	{region "============= 進到設定位置  ============="}
	40: // 判斷前進後退
		IF BD_moveDis - FxB_Clamp_Pos > 0 THEN
			// 目標大於現在位置
			o_BD_Clamp_Close	:= FALSE;
			o_BD_Clamp_Open		:= TRUE;
			step_BD_C.Step  := step_BD_C.Step  + 1;
		ELSIF BD_moveDis - FxB_Clamp_Pos < 0 THEN
			// 目標小於現在位置
			o_BD_Clamp_Close	:= TRUE;
			o_BD_Clamp_Open		:= FALSE;
			step_BD_C.Step  := step_BD_C.Step  + 1;
		ELSE
			step_BD_C.Step  := 90;
		END_IF
		
	41: // 設定位置 - 目前位置 (接近0表示位置到達) <= 停止位移補償(移動速度 * 停止時間) 
		IF ABS(BD_moveDis - FxB_Clamp_Pos) <= (ABS(FxB_Clamp_Spd) * 0.1) THEN
			o_BD_Clamp_Close		:= FALSE;
			o_BD_Clamp_Open		:= FALSE;
			step_BD_C.Step  := step_BD_C.Step  + 1;
		END_IF
		
		// 靜止1秒後，標示為功能完成
		tmr106.IN := ABS(FxB_Clamp_Spd) <= 1;
		tmr106.PT := T#1S;
		IF tmr106.Q THEN
			tmr106.IN := FALSE;
			step_BD_C.Step  := step_BD_C.Step  + 1;
		END_IF
			 
	42:
		o_BD_Clamp_Open		:= FALSE;
		o_BD_Clamp_Close	:= FALSE;
		step_BD_C.Step  := step_BD_C.Step  + 1;
			 
	43:
		 step_BD_C.Step  := 90;
	
{endregion}
		
	90:
		BD_moveDis := 0;
		step_BD_C.bDone := TRUE;
		step_BD_C.Step  := 0;
END_CASE

IF o_BD_Clamp_Open THEN
	b_BD_Clamp := FALSE;
END_IF

step_BD_C.bBuzy := step_BD_C.Step > 0 AND step_BD_C.Step < 10000;
step_BD_C.bError := step_BD_C.Step >= 10000;

IF step_BD_C.bError OR step_BD_C.bBuzy THEN
	step_BD_C.bDone := FALSE;
END_IF
END_ACTION

ACTION Step_BD_01_UnClamp:
CASE step_BD_C.Step  OF
	// FxA動作前檢查檢查
	100: // 檢查Group B Z軸位置，需在桁架中間 (Z pos > 500 )
		tmr01.IN := FALSE;
		IF GbZ.pos > 500 OR GbX.fPos < 50 OR NOT Hmi.Jog_UnLimite THEN
			step_BD_C.Step  := step_BD_C.Step  + 1;
		ELSE
			step_BD_C.Step  := step_BD_C.Step  + 10000;
			strmem1.WRITE(name);
			strmem1.APPEND(":Group B 位置錯誤,再非安全位置:");
			strmem1.APPEND(STR := WCONCAT("(X:", TO_WSTRING(GbX.pos)));
			strmem1.APPEND(STR := WCONCAT(",Y:", TO_WSTRING(GbY.pos)));
			strmem1.APPEND(STR := WCONCAT(",Z:", TO_WSTRING(GbZ.pos)));
			strmem1.APPEND(")");
			pMsg.Push_Error(strmem1.READ);
		END_IF
		
	101: 
		IF o_Oil_Pressure_Pump THEN
			step_BD_C.Step  := step_BD_C.Step  + 1;
		END_IF
		
	102:
		step_BD_C.Step  := 110;
	
		// 確認BD下壓位置
//		IF pressureB_home_sensor AND pressureD_home_sensor THEN
//			step_BD_C.Step  := step_BD_C.Step  + 1;
//		ELSE
//			step_BD_C.Step  := step_BD_C.Step  + 10000;
//			pMsg.Push_Error(StrConcat_2(name, ":下壓B or 下壓D 未停在原點，動作取消 "));
//		END_IF
		
		
		
	110: // 放開選擇
		o_BD_Encoder_enable		:= FALSE;
		o_BD_Encoder_disable	:= TRUE;
		IF BD_moveDis = 0 THEN
			// 退到原點
			step_BD_C.Step  := 120; 
		ELSE
			// 退到設定距離
			step_BD_C.Step  := 140;
		END_IF

	{region "============= 退到原點  ============="}
	120: // 放開BD夾輪夾
		o_BD_Clamp_Close	:= FALSE;
		o_BD_Clamp_Open		:= TRUE;
		step_BD_C.Step  := step_BD_C.Step  + 1;
		
	121: // 確定BD夾輪停止移動
		tmr106.IN := ABS(FxB_Clamp_Spd) <= 1 ;
		tmr106.PT := T#1S;
		IF tmr106.Q THEN
			tmr106.IN := FALSE;
			step_BD_C.Step  := step_BD_C.Step  + 1;
		END_IF
		
	122:
		o_BD_Clamp_Open		:= FALSE;
		step_BD_C.Step  := step_BD_C.Step  + 1;
		
	123: 
		step_BD_C.Step  := 130;
		
	130:
		step_BD_C.Step  := 190;
	{endregion}		
		
		
		
	{region "============= 退到設定距離  ============="}
	140: // 紀錄開始位置
		BD_StartPos := FxB_Clamp_Pos;
		step_BD_C.Step  := step_BD_C.Step  + 1;
		
	141: // 開始後退
		o_BD_Clamp_Close	:= FALSE;
		o_BD_Clamp_Open		:= TRUE;
		step_BD_C.Step := step_BD_C.step + 1;
		
	142: // 大於設定距離
		IF ABS(BD_StartPos - FxB_Clamp_Pos)  >= ABS(BD_moveDis) - ( ABS(FxB_Clamp_Spd) * 0.1) THEN
			o_BD_Clamp_Open		:= FALSE;
			step_BD_C.step := step_BD_C.step + 1;
		END_IF
		
		tmr106.IN := ABS(FxB_Clamp_Spd) <= 1 ;
		tmr106.PT := T#1S;
		IF tmr01.Q THEN
			tmr106.IN := FALSE;
			step_BD_C.Step  := step_BD_C.Step  + 1;
		END_IF
			 
	143:
		o_BD_Clamp_Open		:= FALSE;
		o_BD_Clamp_Close	:= FALSE;
		step_BD_C.step := step_BD_C.step + 1;
			 
	144:
		 step_BD_C.step := 190;
	
	{endregion}
	190:
		o_BD_Encoder_enable		:= FALSE;
		o_BD_Encoder_disable	:= FALSE;
		o_BD_Clamp_Open		:= FALSE;
		step_BD_C.bDone := TRUE;
		step_BD_C.step := 0;
END_CASE
END_ACTION

ACTION Step_BD_02_Stop:
CASE step_BD_C.step OF
	// FxA動作前檢查檢查
	200: 
		step_BD_C.step := 210;
		
		
	210: // BD夾輪夾
		o_BD_Clamp_Open		:= FALSE;
		o_BD_Clamp_Close	:= FALSE;
		step_BD_C.step := step_BD_C.step + 1;
		
	211: 
		step_BD_C.step := 0;
END_CASE
END_ACTION

ACTION Step_BD_03_Home:
CASE step_BD_C.Step  OF
	// FxA動作前檢查檢查
	300:  // 檢查Group B Z軸位置，需在桁架中間 (Z pos > 500 )
		tmr01.IN := FALSE;
		Axis.Encoder_FxA_Clamp.MDP5001_511_Output.MDP5001_511_Control.Set_counter_on_latch_C := FALSE;
		Axis.Encoder_FxA_Clamp.MDP5001_511_Output.MDP5001_511_Control.Set_counter := FALSE;
		IF GbZ.fPos >= 490 OR GbX.fPos < 50 OR Hmi.Jog_UnLimite THEN
			step_BD_C.Step  := step_BD_C.Step  + 1;
		ELSE
			step_BD_C.Step  := step_BD_C.Step  + 20000;
			strmem1.WRITE(name);
			strmem1.APPEND(":Group B 位置錯誤,再非安全位置:");
			strmem1.APPEND(STR := WCONCAT("(X:", TO_WSTRING(GbX.pos)));
			strmem1.APPEND(STR := WCONCAT(",Y:", TO_WSTRING(GbY.pos)));
			strmem1.APPEND(STR := WCONCAT(",Z:", TO_WSTRING(GbZ.pos)));
			strmem1.APPEND(")");
			pMsg.Push_Error(strmem1.READ);
		END_IF
		
		// 確認AC下壓位置
//		IF pressureA_home_sensor AND pressureC_home_sensor THEN
//			step_BD_C.Step  := step_BD_C.Step  + 1;
//		ELSE
//			step_BD_C.Step  := step_BD_C.Step  + 10000;
//			pMsg.Push_Error(StrConcat_2(name, ":下壓A or 下壓C 未停在原點，動作取消 "));
//		END_IF
		
	301: 
		IF o_Oil_Pressure_Pump THEN
			step_BD_C.Step  := step_BD_C.Step  + 1;
		END_IF
		
	302:
		IF IO.i510 THEN
			step_BD_C.Step  := 310; 
		ELSE
			step_BD_C.Step  := 320; 
		END_IF
		
		
		
	310: // AC夾輪夾
		o_BD_Clamp_Open		:= TRUE;
		o_BD_Clamp_Close	:= FALSE;
		step_BD_C.Step  := step_BD_C.Step  + 1;
		
	311:
		tmr106.IN := NOT IO.i510;
		tmr106.PT := T#1S;
		IF tmr106.Q THEN
			tmr106.IN := FALSE;
			step_BD_C.Step  := step_BD_C.Step  + 1;
		END_IF
		
	312:
		o_BD_Clamp_Open		:= FALSE;
		o_BD_Clamp_Close	:= FALSE;
		step_BD_C.Step  := step_BD_C.Step  + 1;
		
	313:
		step_BD_C.Step  := 320;
		
		
	320:
		Axis.Encoder_FxB_Clamp.MDP5001_511_Output.MDP5001_511_Control.Set_counter_on_latch_C := TRUE;
		Axis.Encoder_FxB_Clamp.MDP5001_511_Output.MDP5001_511_Set_counter_value := 10000;
		step_BD_C.Step  := step_BD_C.Step  + 1;
		
	321:
		o_BD_Clamp_Open		:= FALSE;
		o_BD_Clamp_Close	:= TRUE;
		step_BD_C.Step  := step_BD_C.Step  + 1;
			
	322:
		// 編碼器歸零完成
		IF Axis.Encoder_FxB_Clamp.MDP5001_511_Input.MDP5001_511_Status.Set_counter_done THEN
			Axis.Encoder_FxB_Clamp.MDP5001_511_Output.MDP5001_511_Control.Set_counter_on_latch_C := FALSE;
			b_BD_HOME := TRUE;
			step_BD_C.Step  := step_BD_C.Step  + 1;
		END_IF

	323:
		o_BD_Clamp_Open		:= FALSE;
		o_BD_Clamp_Close	:= FALSE;
		step_BD_C.Step  := step_BD_C.Step  + 1;
		
		
	324:
		step_BD_C.Step  := 330;
	
	330:
		o_BD_Clamp_Open		:= TRUE;
		o_BD_Clamp_Close	:= FALSE;
		step_BD_C.Step  := step_BD_C.Step  + 1;
		
	331:
		tmr106.IN := NOT IO.i510;
		tmr106.PT := T#1S;
		IF tmr106.Q THEN
			tmr106.IN := FALSE;
			step_BD_C.Step  := step_BD_C.Step  + 1;
		END_IF
		
	332:
		o_BD_Clamp_Open		:= FALSE;
		o_BD_Clamp_Close	:= FALSE;
		step_BD_C.Step  := step_BD_C.Step  + 1;
		
	333:
		step_BD_C.bDone := TRUE;
		step_BD_C.Step  := 0;
		
END_CASE
END_ACTION

ACTION Step_C_Push_UnPush:
CASE step_C_P.Step OF
(*	================================
				C下壓
 	================================*)	

	// FxA動作前檢查檢查
	1: // 檢查Group B Z軸位置，需在桁架中間 (Z pos > 500 )
		step_C_P.Step  := step_C_P.Step  + 1;
// 		IF GbZ.fPos >= 495 OR GbX.fPos > 50 OR Hmi.Jog_UnLimite THEN
// 			step_C_P.Step  := step_C_P.Step  + 1;
// 		ELSE
// 			step_C_P.Step  := step_C_P.Step  + 10000;
// 			strmem1.WRITE(name);
// 			strmem1.APPEND(".C_Push");
// 			strmem1.APPEND(":Group B 位置錯誤,再非安全位置:");
// 			strmem1.APPEND(STR := WCONCAT("(X:", TO_WSTRING(GbX.pos)));
// 			strmem1.APPEND(STR := WCONCAT(",Y:", TO_WSTRING(GbY.pos)));
// 			strmem1.APPEND(STR := WCONCAT(",Z:", TO_WSTRING(GbZ.pos)));
// 			strmem1.APPEND(")");
// 			pMsg.Push_Error(strmem1.READ);
// 		END_IF
		
	2:
		tmr114.IN := TRUE;
		tmr114.PT := T#10S;
		IF o_Oil_Pressure_Pump OR tmr113.Q THEN
			tmr113.IN := FALSE;
			IF o_Oil_Pressure_Pump THEN
				step_C_P.Step  := step_C_P.Step  + 1;
			ELSIF tmr113.Q THEN
				pMsg.Push_Error(WStrConcat(name, ".C_Push:下壓B等待油壓系統啟動逾時"));
				step_C_P.Step  := step_C_P.Step  + 10000;
			END_IF
		END_IF
		
	3:
		tmr103.IN := FALSE;
		tmr113.IN := FALSE;
		step_C_P.Step  := 10;
		
		
	10: // 下壓啟動
		o_PressureC_Up := FALSE;
		o_PressureC_Dn := TRUE;
		step_C_P.Step  := step_C_P.Step  + 1;
		
	11:
		tmr103.IN := TRUE;
		tmr103.PT := T#500MS;
		IF tmr103.q THEN
			tmr103.IN := FALSE;
			step_C_P.Step  := step_C_P.Step  + 1;
		END_IF
		
	12:
// 		o_PressureC_Dn := FALSE;
		step_C_P.Step  := step_C_P.Step  + 1;
		
	13:
		tmr103.IN := pressureC_pressure_sensor;
		tmr103.PT := T#500MS;
		tmr113.IN := TRUE;
		tmr113.PT := T#30S;
		IF tmr103.q OR tmr113.q THEN
			tmr103.IN := FALSE;
			tmr113.IN := FALSE;
			step_C_P.Step  := step_C_P.Step  + 1;
		END_IF
		
	14:
		step_C_P.bDone := TRUE;
		step_C_P.Step  := 0;


(*	================================
				C放開
 	================================*)
	// FxA動作前檢查檢查
	100: // 檢查Group B Z軸位置，需在桁架中間 (Z pos > 500 )
		IF GbZ.pos >= 495 OR GbX.fPos < 50 OR Hmi.Jog_UnLimite OR
			(_C_UnPush_Time > 0 AND _C_UnPush_Time < 10) THEN
			step_C_P.Step  := step_C_P.Step  + 1;
		ELSE
			step_C_P.Step  := step_C_P.Step  + 10000;
			strmem1.WRITE(name);
			strmem1.APPEND(".C_Push");
			strmem1.APPEND(":Group B 位置錯誤,再非安全位置:");
			strmem1.APPEND(STR := WCONCAT("(X:", TO_WSTRING(GbX.pos)));
			strmem1.APPEND(STR := WCONCAT(",Y:", TO_WSTRING(GbY.pos)));
			strmem1.APPEND(STR := WCONCAT(",Z:", TO_WSTRING(GbZ.pos)));
			strmem1.APPEND(")");
			pMsg.Push_Error(strmem1.READ);
		END_IF
		
	101:
		IF o_Oil_Pressure_Pump OR tmr113.Q THEN
			tmr113.IN := FALSE;
			IF o_Oil_Pressure_Pump THEN
				step_C_P.Step  := step_C_P.Step  + 1;
			ELSIF tmr113.Q THEN
				pMsg.Push_Error(WStrConcat(name, ".C_Push:下壓B等待油壓系統啟動逾時"));
				step_C_P.Step  := step_C_P.Step  + 10000;
			END_IF
		END_IF
		
	102:
		tmr103.IN := FALSE;
		tmr113.IN := FALSE;
		step_C_P.Step  := 110;
		
		
	110: // 放開啟動
		o_PressureC_Up := TRUE;
		o_PressureC_Dn := FALSE;
		IF _C_UnPush_Time > 0 THEN
			// 微上升
			step_C_P.Step  := step_C_P.Step  + 20;
		ELSE
			// 升回原點
			step_C_P.Step  := step_C_P.Step  + 10;
		END_IF
		
(*	========================================
					升回原點
	========================================	*)
	120:
		tmr103.IN := TRUE;
		tmr103.PT := T#500MS;
		IF tmr103.q THEN
			tmr103.IN := FALSE;
			step_C_P.Step  := step_C_P.Step  + 1;
		END_IF
		
	121:
// 		o_PressureC_Up := FALSE;
		step_C_P.Step  := step_C_P.Step  + 1;
		
	122:
		tmr103.IN := pressureC_home_sensor;
		tmr103.PT := T#500MS;
		tmr113.IN := TRUE;
		tmr113.PT := T#10S;
		IF tmr103.q OR tmr113.q THEN
			tmr103.IN := FALSE;
			tmr113.IN := FALSE;
			o_PressureC_Up := FALSE;
			step_C_P.Step  := step_C_P.Step  + 1;
		END_IF
		
	123:
		step_C_P.bDone := TRUE;
		step_C_P.Step  := 0;

(*	========================================
					微上升
	========================================	*)
	
	130:
		tmr103.IN := TRUE;
		tmr103.PT := TO_TIME(_C_UnPush_Time * 100);
		IF tmr103.q THEN
			tmr103.IN := FALSE;
			step_C_P.Step  := step_C_P.Step  + 1;
		END_IF
		
	131:
		o_PressureC_Up := FALSE;
		step_C_P.Step  := step_C_P.Step  + 1;
		
	132:
		step_C_P.bDone := TRUE;
		step_C_P.Step  := 0;
	
END_CASE

step_C_P.bBuzy := step_C_P.Step  > 0 AND step_C_P.Step  < 10000;
step_C_P.bError := step_C_P.Step  >= 10000;

IF step_C_P.bBuzy OR step_C_P.bError THEN
	step_C_P.bDone := FALSE;
END_IF
END_ACTION

ACTION Step_D_Push_UnPush:
CASE step_D_P.Step  OF
(*	================================
				D下壓
 	================================*)	

	// FxA動作前檢查檢查
	1: // 檢查Group B Z軸位置，需在桁架中間 (Z pos > 500 )
		IF GbZ.fPos >= 495 OR GbX.fPos < 50 OR Hmi.Jog_UnLimite THEN
			step_D_P.Step  := step_D_P.Step  + 1;
		ELSE
			step_D_P.Step  := step_D_P.Step  + 10000;
			strmem1.WRITE(name);
			strmem1.APPEND(":Group B 位置錯誤,再非安全位置:");
			strmem1.APPEND(STR := WCONCAT("(X:", TO_WSTRING(GbX.pos)));
			strmem1.APPEND(STR := WCONCAT(",Y:", TO_WSTRING(GbY.pos)));
			strmem1.APPEND(STR := WCONCAT(",Z:", TO_WSTRING(GbZ.pos)));
			strmem1.APPEND(")");
			pMsg.Push_Error(strmem1.READ);
		END_IF
		
	2:
		tmr114.IN := TRUE;
		tmr114.PT := T#10S;
		IF o_Oil_Pressure_Pump OR tmr114.Q THEN
			tmr114.IN := FALSE;
			IF o_Oil_Pressure_Pump THEN
				step_D_P.Step  := step_D_P.Step  + 1;
			ELSIF tmr114.Q THEN
				pMsg.Push_Error(WStrConcat(name, ".C_Push:下壓B等待油壓系統啟動逾時"));
				step_D_P.Step  := step_D_P.Step  + 10000;
			END_IF
		END_IF
		
	3:
		tmr104.IN := FALSE;
		tmr114.IN := FALSE;
		step_D_P.Step  := 10;
		
		
	10: // 下壓啟動
		o_PressureD_Up := FALSE;
		o_PressureD_Dn := TRUE;
		step_D_P.Step  := step_D_P.Step  + 1;
		
	11:
		tmr104.IN := TRUE;
		tmr104.PT := T#500MS;
		IF tmr104.q THEN
			tmr104.IN := FALSE;
			step_D_P.Step  := step_D_P.Step  + 1;
		END_IF
		
	12: // 改三位閥，須持續送
// 		o_PressureD_Dn := FALSE;
		step_D_P.Step  := step_D_P.Step  + 1;
		
	13:
		tmr104.IN := pressureD_pressure_sensor;
		tmr104.PT := T#500MS;
		tmr114.IN := TRUE;
		tmr114.PT := T#30S;
		IF tmr104.q OR tmr114.q THEN
			tmr104.IN := FALSE;
			tmr114.IN := FALSE;
			step_D_P.Step  := step_D_P.Step  + 1;
		END_IF
		
	14:
		step_D_P.bDone := TRUE;
		step_D_P.Step  := 0;


(*	================================
				D放開
 	================================*)
	// FxA動作前檢查檢查
	100: // 檢查Group B Z軸位置，需在桁架中間 (Z pos > 500 )
		IF GbZ.fPos >= 495 OR GbX.fPos < 50 OR Hmi.Jog_UnLimite OR 
			(_D_UnPush_Time > 0 AND _D_UnPush_Time < 10) THEN
			step_D_P.Step  := step_D_P.Step  + 1;
		ELSE
			step_D_P.Step  := step_D_P.Step  + 10000;
			strmem1.WRITE(name);
			strmem1.APPEND(".D_Push");
			strmem1.APPEND(":Group B 位置錯誤,再非安全位置:");
			strmem1.APPEND(STR := WCONCAT("(X:", TO_WSTRING(GbX.pos)));
			strmem1.APPEND(STR := WCONCAT(",Y:", TO_WSTRING(GbY.pos)));
			strmem1.APPEND(STR := WCONCAT(",Z:", TO_WSTRING(GbZ.pos)));
			strmem1.APPEND(")");
			pMsg.Push_Error(strmem1.READ);
		END_IF
		
	101:
		IF o_Oil_Pressure_Pump OR tmr114.Q THEN
			tmr114.IN := FALSE;
			IF o_Oil_Pressure_Pump THEN
				step_D_P.Step  := step_D_P.Step  + 1;
			ELSIF tmr114.Q THEN
				pMsg.Push_Error(WStrConcat(name, ".D_Push:下壓D等待油壓系統啟動逾時"));
				step_D_P.Step  := step_D_P.Step  + 10000;
			END_IF
		END_IF
		
	102:
		tmr104.IN := FALSE;
		tmr114.IN := FALSE;
		step_D_P.Step  := 110;
		
		
	110: // 放開啟動
		o_PressureD_Up := TRUE;
		o_PressureD_Dn := FALSE;
		IF _D_UnPush_Time > 0 THEN
			// 微上升
			step_D_P.Step  := step_D_P.Step  + 20;
		ELSE
			// 升回原點
			step_D_P.Step  := step_D_P.Step  + 10;
		END_IF
		
(*	========================================
					升回原點
	========================================	*)
	120: // 升回原點
		tmr104.IN := TRUE;
		tmr104.PT := T#500MS;
		IF tmr104.q THEN
			tmr104.IN := FALSE;
			step_D_P.Step  := step_D_P.Step  + 1;
		END_IF
		
	121: // 改三位閥，須持續送
// 		o_PressureD_Up := FALSE;
		step_D_P.Step  := step_D_P.Step  + 1;
		
	122:
		tmr104.IN := pressureD_home_sensor;
		tmr104.PT := T#500MS;
		tmr114.IN := TRUE;
		tmr114.PT := T#30S;
		IF tmr104.q OR tmr114.q THEN
			tmr104.IN := FALSE;
			tmr114.IN := FALSE;
			o_PressureD_Up := FALSE;
			step_D_P.Step  := step_D_P.Step  + 1;
		END_IF
		
	123:
		step_D_P.bDone := TRUE;
		step_D_P.Step  := 0;

(*	========================================
					微上升
	========================================	*)
	130:
		tmr104.IN := TRUE;
		tmr104.PT := TO_TIME(_D_UnPush_Time * 100);
		IF tmr104.q THEN
			tmr104.IN := FALSE;
			step_D_P.Step  := step_D_P.Step  + 1;
		END_IF
		
	131:
		o_PressureD_Up := FALSE;
		step_D_P.Step  := step_D_P.Step  + 1;
		
	132:
		step_D_P.bDone := TRUE;
		step_D_P.Step  := 0;
		
END_CASE

step_D_P.bBuzy := step_D_P.Step  > 0 AND step_D_P.Step  < 10000;
step_D_P.bError := step_D_P.Step  >= 10000;

IF step_D_P.bBuzy OR step_D_P.bError THEN
	step_D_P.bDone := TRUE;
END_IF
END_ACTION

ACTION timer:
tmr01();
tmr02();

tmr101();
tmr102();
tmr103();
tmr104();
tmr105();
tmr106();

tmr111();
tmr112();
tmr113();
tmr114();
tmr115();
tmr116();

tmr_wdt();
END_ACTION

END_PROGRAM

// ---- POUs/功能塊/字串處理功能塊/字串記憶/WStrMem.TcPOU
FUNCTION_BLOCK WStrMem
VAR_INPUT
END_VAR
VAR_OUTPUT
END_VAR
VAR
	mem : WSTRING;
END_VAR

METHOD APPEND : BOOL
VAR_INPUT
	STR : WSTRING;
END_VAR
mem := WCONCAT(mem , STR);
END_METHOD

METHOD INSERT : BOOL
VAR_INPUT
	STR : WSTRING;
END_VAR
mem := WCONCAT(STR, mem);
END_METHOD

PROPERTY READ : WSTRING
GET
READ := mem;
END_GET
END_PROPERTY

METHOD WRITE : BOOL
VAR_INPUT
	STR :WSTRING;
END_VAR
mem := STR;
END_METHOD

END_FUNCTION_BLOCK

// ---- POUs/功能塊/pMsg.TcPOU
PROGRAM pMsg
VAR
	msg: MsgPush;
END_VAR

METHOD PUBLIC Push_Alarm : BOOL
VAR_INPUT
	STR : WSTRING;
END_VAR
msg.iMessageId := 0;
msg.msgeLevel := MsgLevel.Alarm;
msg.sMessageStr1:=STR;
msg();
IF hmi.State = MachineState.Auto_mode THEN
	Safety.SystemAlarm := TRUE;
end_if
END_METHOD

METHOD PUBLIC Push_Alarm_NoPause : BOOL
VAR_INPUT
	STR : WSTRING;
	STR1 : WSTRING := "";
	STR2 : WSTRING := "";
	STR3 : WSTRING := "";
	STR4 : WSTRING := "";
	STR5 : WSTRING := "";
END_VAR
msg.iMessageId := 0;
msg.msgeLevel := MsgLevel.Alarm;
msg.sMessageStr1:=str;
msg.sMessageStr1:=WCONCAT(STR1:= msg.sMessageStr1, STR2:= STR1);
msg.sMessageStr1:=WCONCAT(STR1:= msg.sMessageStr1, STR2:= STR2);
msg.sMessageStr1:=WCONCAT(STR1:= msg.sMessageStr1, STR2:= STR3);
msg.sMessageStr1:=WCONCAT(STR1:= msg.sMessageStr1, STR2:= STR4);
msg.sMessageStr1:=WCONCAT(STR1:= msg.sMessageStr1, STR2:= STR5);
msg();
END_METHOD

METHOD PUBLIC Push_Error : BOOL
VAR_INPUT
	STR : WSTRING;
END_VAR
msg.iMessageId := 0;
msg.msgeLevel := MsgLevel.Error;
msg.sMessageStr1:=STR;
SystemError := TRUE;
hmi.State := MachineState.error;
msg();
END_METHOD

METHOD PUBLIC Push_Info : BOOL
VAR_INPUT
	STR : WSTRING;
	
END_VAR
msg.iMessageId := 0;
msg.msgeLevel := MsgLevel.Info;
msg.sMessageStr1:=STR;
msg();
END_METHOD

END_PROGRAM

// ---- MSG/通知訊息/MsgPush.TcPOU
FUNCTION_BLOCK MsgPush
VAR_INPUT
	// 事件等級(MessageLevel.info:訊息、.Alarm:警告、.Error:錯誤)
	msgeLevel: MsgLevel;
	// 訊息編號
	iMessageId: UINT;
	// 訊息插入文字1
	sMessageStr1: WSTRING(80) := "";
	// 訊息插入文字2
	sMessageStr2: WSTRING(80) := "";
	
END_VAR

VAR
	msg		: MsgStruct;
	
	MsgNum			: USINT;
END_VAR
VAR_OUTPUT
	bDone: BOOL;
	nState : INT;
END_VAR

MsgNum := ULINT_TO_USINT(MsgBuff.evenNumber MOD 16);



//MsgBuff.messageList[MsgNum].MsgTime := 	FILETIME_TO_DT(currentTime);
//MsgBuff.messageList[MsgNum].Level :=	msgeLevel;
//MsgBuff.messageList[MsgNum].Number :=	iMessageId;
//MsgBuff.messageList[MsgNum].MsgStr1 :=	sMessageStr1;
//MsgBuff.messageList[MsgNum].MsgStr2 :=	sMessageStr2;
//MsgBuff.messageList[MsgNum].Sn :=		MsgBuff.evenNumber;
MsgBuff.evenNumber := MsgBuff.evenNumber + 1;

bDone := FALSE;

msg.MsgTime := 	msgbuff.currentTime;
msg.Level :=	msgeLevel;
msg.Number :=	iMessageId;
msg.MsgStr1 :=	sMessageStr1;
msg.MsgStr2 :=	sMessageStr2;
msg.raw_msg_str := sMessageStr1;

MsgBuff.messageList[MsgNum] := msg;

END_FUNCTION_BLOCK

// ---- POUs/功能塊/字串處理功能塊/字串連接/WStrConcat.TcPOU
FUNCTION WStrConcat : WSTRING(511)
VAR_INPUT
	str0 : WSTRING(511) := "";
	str1 : WSTRING(511) := "";
	str2 : WSTRING(511) := "";
	str3 : WSTRING(511) := "";
	str4 : WSTRING(511) := "";
	str5 : WSTRING(511) := "";
	str6 : WSTRING(511) := "";
	str7 : WSTRING(511) := "";
	str8 : WSTRING(511) := "";
END_VAR
VAR
	tmpstr : WSTRING(511);
END_VAR

tmpstr := WCONCAT(STR1:= str0, STR2:= str1);
tmpstr := WCONCAT(STR1:= tmpstr, STR2:= str2);
tmpstr := WCONCAT(STR1:= tmpstr, STR2:= str3);
tmpstr := WCONCAT(STR1:= tmpstr, STR2:= str4);
tmpstr := WCONCAT(STR1:= tmpstr, STR2:= str5);
tmpstr := WCONCAT(STR1:= tmpstr, STR2:= str6);
tmpstr := WCONCAT(STR1:= tmpstr, STR2:= str7);
tmpstr := WCONCAT(STR1:= tmpstr, STR2:= str8);
WStrConcat := tmpstr;
RETURN;

END_FUNCTION

// ---- POUs/動作流程控制/AxisGroup功能塊/GroupA.TcPOU
PROGRAM GroupA
VAR
	step		: INT;
	
	StepA		: Sub_Step;
	
	// X軸映射
	Ax : I_Axis;
	Axs: Sub_Step;
	// Y軸映射
	Ay : I_Axis;
	Ays: Sub_Step;
	// X軸映射
	Az : I_Axis;
	Azs: Sub_Step;
	
	Ax_P_Limite : LREAL;
	Ax_N_Limite : LREAL;
	Ay_P_Limite : LREAL;
	Ay_N_Limite : LREAL;
	Az_P_Limite : LREAL;
	Az_N_Limite : LREAL;
	
	
	// 移動命令的 X位置
	moveCmd_X: LREAL;
	// 移動命令的 Y位置
	moveCmd_Y: LREAL;
	// 移動命令 速度
	moveCmd_Spd: LREAL;
	
	moveZdis	: REAL;
	tmr01A		: TON;
	tmr01		: TON;
	tmr02		: TON;
	
	// 坐標系的參考原點
	pointRef : XYZ_Point;
	
	// 移動位置X 計算結果
	tmpPos_X: LREAL;
	// 移動位置Y 計算結果
	tmpPos_Y: LREAL;
	
	
	// 雷射圖形移動距離 Y
	Dxf_Y_Move : LREAL;

	// 測量到的Z位置
	z_PosMeasure: REAL;
	
	// 距離感應器IO
	DisSensor_SSC1: BOOL;
	// 距離感應器距離
	DisSensor_Dis: REAL;
	
	Boot : BOOL := TRUE;
	
	
	// 執行中的清單號
	WorkNum: INT;
	
	// 鏡頭 吹氣
	q_Lens_Blow :BOOL;
	
	// 重試計數器
	_retryCnt: INT;
	
	// 可以開始雕刻 (Fx就緒)
	_ReadyToPrint :BOOL;
	// 可以開始移動 (Fx就緒)
	_ReadyToMove :BOOL;
	
	
	// 計算上次打油後的一棟距離
	X_Move: LREAL;
	Y_Move: LREAL;
	Z_Move: LREAL;
	tmr_oil: TON;
	
	_log : Step_Log; 
	_logA : Step_Log; 
	sql_hand: UDINT;
END_VAR
VAR_INPUT

END_VAR
VAR_OUTPUT
	// 工件高度
	Size_H : REAL;
	// 工件座標
	RefPos : XYZ_Point;
	
	// 功能執行中
	bBuzy 	: BOOL;
	// 功能結束
	bDone	: BOOL;
	// 發生錯誤
	bError	: BOOL;
END_VAR

IF Boot THEN
	Ax := axis.GaX;
	Ay := axis.GaY;
	Az := axis.GaZ;
	boot := FALSE;
END_IF

Axs := Ax.State;
Ays := Ay.State;
Azs := Az.State;

Ax_P_Limite := posc.GaX_P_Limite;
Ax_N_Limite := posc.GaX_N_Limite;
Ay_P_Limite := posc.GaY_P_Limite;
Ay_N_Limite := posc.GaY_N_Limite;
Az_P_Limite := posc.GaZ_P_Limite;
Az_N_Limite := posc.GaZ_N_Limite;

DisSensor_SSC1	:= Sensor.sensorA.SSC1_1;
DisSensor_Dis	:= Sensor.sensorA.Distance;

IF (EStop OR SystemError) THEN
	IF bBuzy THEN
		step := step  + 10000;
	END_IF
	IF StepA.bBuzy THEN
		StepA.step := StepA.step  + 10000;
	END_IF
	Hmi_Web.Process_Data_UUID_A_Start := FALSE;
	q_Lens_Blow := FALSE;
END_IF

bBuzy := step > 0 AND step < 10000;
bError := step >= 10000;
IF bBuzy OR bError THEN
	bDone := FALSE;
END_IF

Step_01_DoPayloadList();
Step_02_Do_2nd_in_list();
Step_03_DoLaserAction();

StepA.bBuzy := StepA.step > 0 AND StepA.step < 10000;
StepA.bError := StepA.step >= 10000;
IF StepA.bBuzy OR StepA.bError THEN
	StepA.bDone := FALSE;
END_IF

Step_A_01_MoveToXY();
Step_A_02_FindZ();
Step_A_03_FindY();
Step_A_10_MoveToXY_REF();
Step_A_20_ToStanbyPos();

Timer();

RefPos.X := GaX.Pos - pointRef.X;
RefPos.Y := GaY.Pos - pointRef.Y;
RefPos.Z := GaZ.Pos - pointRef.Z;

ProjectData.Now_Steel_Payload_A_DataNumber_Done := WorkNum;

io.q305 := q_Lens_Blow;

_log(name:= 'GroupA', step:= step);
_logA(name:= 'GroupA_Mov', step:= StepA.Step);

METHOD Do_WorkList : BOOL
VAR_INPUT
END_VAR
bDone := FALSE;


_log.fbJson.StartObject();
_log.fbJson.AddKeyString('MethodName','Do_WorkList');
_log.JsonOutput();


Step := 100;
END_METHOD

METHOD FindZ : BOOL
VAR_INPUT
END_VAR
StepA.bDone := FALSE;


// ============ 紀錄啟動條件 ============
_logA.fbJson.StartObject();
_logA.fbJson.AddKeyString('MethodName','FindZ');
_logA.JsonOutput();
// ======================================


StepA.step := 200;
END_METHOD

METHOD FindZ_Fast : BOOL
VAR_INPUT
END_VAR
StepA.bDone := FALSE;


// ============ 紀錄啟動條件 ============
_logA.fbJson.StartObject();
_logA.fbJson.AddKeyString('MethodName','FindZ');
_logA.JsonOutput();
// ======================================



StepA.step := 230;
END_METHOD

ACTION Oil:
X_Move := Axis.GaX_total_Move - Axis.GaX_Last_Oil;
Y_Move := Axis.GaY_total_Move - Axis.GaY_Last_Oil;
Z_Move := Axis.GaZ_total_Move - Axis.GaZ_Last_Oil;

IF X_Move > 1000000 OR Y_Move > 1000000 OR Z_Move > 1000000 THEN
	IO.q204 := TRUE;
END_IF
END_ACTION

PROPERTY ReadyToMove : BOOL
GET
ReadyToMove := _ReadyToMove;
END_GET
SET
_ReadyToMove := ReadyToMove;
END_SET
END_PROPERTY

PROPERTY ReadyToPrint : BOOL
GET
ReadyToPrint := _ReadyToPrint;
END_GET
SET
_ReadyToPrint := ReadyToPrint;
END_SET
END_PROPERTY

METHOD Set_X_Ref
VAR_INPUT
	Value : LREAL;
END_VAR
pointRef.X := Value;
END_METHOD

METHOD Set_Y_Ref
VAR_INPUT
	Value : LREAL;
END_VAR
pointRef.Y := Value;
END_METHOD

ACTION Step_01_DoPayloadList:
CASE step OF
(*	===============================================
		開始做 Payload_A_Data_buff 清單內的工作
	===============================================*)
	100: // 以數量判斷是否有工作
		WorkNum := 0;		// 初始化工作暫存器
		IF ProjectData.Now_Steel_Payload_A_DataNumber > 0 THEN
			step := step + 1;
		ELSE
		// 沒有這個軸向的工作，直接送出完成
			bDone := TRUE;
			Step := 0;
		END_IF
 
			
	101:
		Hmi_Web.Process_Data_UUID_C_Start := FALSE;
		step := 110;
		
(*	===============================================
					設定工作中的專案
	===============================================*)
	110:
		ProjectData.Payload_A_Data_Now := ProjectData.Payload_A_Data_buff[WorkNum];
		Hmi_Web.Process_Data_UUID_C := ProjectData.Payload_A_Data_buff[WorkNum].data_uid;
		step := step + 1;
	
	111:
		step := 120;
		
(*	===============================================
					移動到位置
	===============================================*)
	120:
		IF _ReadyToMove THEN
			step := step + 1;
		END_IF
		
	121:
		XY_Move_Ref(
			ProjectData.Payload_A_Data_Now.Point_X, 
			ProjectData.Payload_A_Data_Now.Point_Y, 
			SpdC.HighSpeed
		);
		step := step + 1;
		
	122:
		IF stepA.bBuzy OR stepA.bError THEN
			step := step + 1;
		END_IF
		
	123:
		IF stepA.bDone THEN
			step := step + 1;
		ELSIF stepA.bError THEN
			step := step + 10000;
		END_IF
		
	124:
		step := 130;
	

(*	===============================================
				雷射主機 啟動 預覽/雕刻 動作
	===============================================*)	
	130:
		step := 300;
END_CASE
END_ACTION

ACTION Step_02_Do_2nd_in_list:
CASE step OF
	200:
		step := 210;
		
(*	===============================================
					設定工作中的專案
	===============================================*)
	210:
		ProjectData.Payload_A_Data_Now := ProjectData.Payload_A_Data_buff[WorkNum];
		Hmi_Web.Process_Data_UUID_C := ProjectData.Payload_A_Data_buff[WorkNum].data_uid;
		step := step + 1;
	
	211:
		step := 220;
		
(*	===============================================
					移動到位置
	===============================================*)
	220:
		XY_Move_Ref(
			ProjectData.Payload_A_Data_Now.Point_X, 
			ProjectData.Payload_A_Data_Now.Point_Y, 
			SpdC.HighSpeed
		);
		step := step + 1;
		
	221:
		IF stepA.bBuzy OR stepA.bError THEN
			step := step + 1;
		END_IF
		
	222:
		IF stepA.bDone THEN
			step := step + 1;
		ELSIF stepA.bError THEN
			step := step + 10000;
		END_IF
		
	223:
		step := 230;
		
(*	===============================================
				雷射主機 啟動 預覽/雕刻 動作
	===============================================*)	
	230:
		step := 300;
END_CASE
END_ACTION

ACTION Step_03_DoLaserAction:
CASE step OF
	300:
		IF ReadyToPrint THEN
			step := step + 1;
		END_IF
		
	301:
		sql_hand := ReadSQLData.Set_Payload_Start(ProjectData.Payload_A_Data_Now.data_uid);
		IF sql_hand <> 0 THEN
			step := step + 1;
		END_IF
		
	302:
		step := 310;

(*	===============================================
				雷射主機 啟動 預覽/雕刻 動作
	===============================================*)	
	310:
		q_Lens_Blow := TRUE;
		IF LEN(Hmi_Web.Process_Data_UUID_C) = 0 THEN
			Hmi_Web.Process_Data_UUID_C := ProjectData.Payload_A_Data_buff[WorkNum].data_uid;
		ELSE
			step := step + 1;
		END_IF
		
	311:
		Hmi_Web.Process_Data_UUID_C_Start := TRUE;
		// ============ 紀錄啟動條件 ============
		_log.fbJson.StartObject();
		_log.fbJson.AddKeyString('StepName','Laser_A_Start');
		_log.fbJson.AddKeyBool('Process_Data_UUID_C_Start:', Hmi_Web.Process_Data_UUID_C_Start);
		_log.fbJson.AddKeyString('Payload_A_Data_Now', ProjectData.Payload_A_Data_Now.data_uid);
		_log.JsonOutput();
		// ======================================
		step := step + 1;
		
	312:
		tmr01.PT := T#500MS;
		tmr01.IN := TRUE;
		IF tmr01.Q THEN
			tmr01.IN := FALSE;
			tmr02.IN := FALSE;
			step := step + 1;
		END_IF
		
	313:
		tmr01.PT := TO_TIME(MaCfg.LaserPrinter_Timeout);
		tmr01.IN := TRUE;
		tmr02.PT := T#250mS;
		tmr02.IN := NOT Hmi_Web.Process_Data_UUID_C_Start;
		IF tmr02.Q THEN
			Hmi_Web.Process_Data_UUID_C :='';
			tmr01.IN := FALSE;
			tmr02.IN := FALSE;
			// ============ 紀錄啟動條件 ============
			_log.fbJson.StartObject();
			_log.fbJson.AddKeyString('StepName','Laser_A_Done');
			_log.JsonOutput();
			// ======================================
			step := step + 1;
		ELSIF tmr01.Q THEN
			tmr01.IN := FALSE;
			tmr02.IN := FALSE;
			pMsg.Push_Error("GroupA:雷射動作超時");
			step := step + 10000;
		END_IF
		
	314:
		q_Lens_Blow := FALSE;
		WorkNum := WorkNum + 1;
		step := 320;
		
(*	================================================
				開始下個循環或此區域結束
	================================================*)	
	320:
		sql_hand := ReadSQLData.Set_Payload_Finish(ProjectData.Payload_A_Data_Now.data_uid);
		IF sql_hand <> 0 THEN
			step := step + 1;
		END_IF
	
	321:
		IF WorkNum < ProjectData.Now_Steel_Payload_A_DataNumber THEN
		// 這個區域還有工作
			step := step + 1;
		ELSE
		// 這個區域工作結束
			step := 390;
		END_IF
		
	322:
		// 設定工作中的專案
		step := 200;
		
(*	================================================
				此區域結束
	================================================*)		
	390:
		bDone := TRUE;
		step := 0;
END_CASE
END_ACTION

ACTION Step_A_01_MoveToXY:
CASE StepA.step OF
	100:
		IF moveCmd_X < Ax_P_Limite AND moveCmd_X > Ax_N_Limite THEN
			StepA.step := StepA.step + 1;
		ELSIF moveCmd_X >= Ax_P_Limite THEN
			StepA.step := StepA.step + 10000;
			pMsg.Push_Alarm("GroupA MoveXY:命令位置超出X軸+極限");
		ELSE
			StepA.step := StepA.step + 10000;
			pMsg.Push_Alarm("GroupA MoveXY:命令位置超出X軸-極限");
		END_IF
 
			
	101:
		IF moveCmd_Y < Ay_P_Limite AND moveCmd_Y > Ay_N_Limite THEN
			StepA.step := StepA.step + 1;
		ELSIF moveCmd_Y >= Ay_P_Limite THEN
			StepA.step := StepA.step + 10000;
			pMsg.Push_Alarm("GroupA MoveXY:命令位置超出Y軸+極限");
		ELSE
			StepA.step := StepA.step + 10000;
			pMsg.Push_Alarm("GroupA MoveXY:命令位置超出Y軸-極限");
		END_IF
		
	102:
		StepA.step := 110;
		
	110:
		Ax.AbsMove(moveCmd_X, moveCmd_Spd);
		Ay.AbsMove(moveCmd_Y, moveCmd_Spd);
		StepA.step := StepA.step + 1;
		
	111:
		IF (Axs.bBuzy OR Axs.bError) AND (Ays.bBuzy OR Ays.bError) THEN
			StepA.step := StepA.step + 1;
		END_IF
		
	112:
		IF Axs.bDone AND Ays.bDone THEN
			StepA.step := StepA.step + 1;
		ELSIF Axs.bError OR Ays.bError THEN
			StepA.step := StepA.step + 10000;
		END_IF
		
	113:
		StepA.bDone := TRUE;
		StepA.step := 0;
		
END_CASE
END_ACTION

ACTION Step_A_02_FindZ:
CASE StepA.step OF
	200: // 判斷當距離再200~400間，
		IF DisSensor_Dis < 200 OR DisSensor_Dis > 400 THEN
			StepA.step := StepA.step + 1;
		ELSE
			StepA.step := 220;
		END_IF
		
	201:
		IF pointRef.Y = 0 THEN
			pointRef.Y := MaCfg.laserA_Y_ReferencePos - ProjectData.Now_Steel.Width;
		END_IF
		StepA.step := 210;
		
		
	210: 
		Az.AbsMove(posc.GaZ_P_Limite - 20, SpdC.HighSpeed);
		StepA.step := StepA.step + 1;
		
	211:
		IF Azs.bBuzy OR Azs.bError THEN
			StepA.step := StepA.step + 1;
		END_IF
		
	212:
		IF Azs.bDone THEN
			StepA.step := StepA.step + 1;
		ELSIF Azs.bError THEN
			StepA.step := StepA.step + 10000;
		END_IF
		
	213:
		StepA.step := 220;
		
	220:
		Ax.AbsMove((macfg.laserA_X_DisSensor2LaserCenter * -1) + 10, SpdC.HighSpeed);
		Ay.AbsMove((ProjectData.Now_Steel.Width / 2) + pointRef.Y, SpdC.HighSpeed);
		StepA.step := StepA.step + 1;
		
	221:
		IF (Axs.bBuzy OR Axs.bError) AND (Ays.bBuzy OR Ays.bError) THEN
			StepA.step := StepA.step + 1;
		END_IF
		
	222:
		IF Axs.bDone AND Ays.bDone THEN
			StepA.step := StepA.step + 1;
		ELSIF Axs.bError OR Ays.bError THEN
			StepA.step := StepA.step + 10000;
		END_IF
		
	223:
		StepA.step := 230;
		
	230:
		IF DisSensor_Dis > 0 THEN
			StepA.step := StepA.step + 1;
		ELSE
			pMsg.Push_Error("GroupA: 測距感應器數值錯誤");
			StepA.step := StepA.step + 10000;
		END_IF
		
	231:
		moveZdis := DisSensor_Dis - Macfg.laserA_Dis;
		StepA.step := StepA.step + 1;
		
	232:
		Az.RelMove(moveZdis * -1, SpdC.HighSpeed);
		StepA.step := StepA.step + 1;
		
	233:
		IF Azs.bBuzy OR Azs.bError THEN
			StepA.step := StepA.step + 1;
		END_IF
		
	234:
		IF Azs.bDone THEN
			StepA.step := StepA.step + 1;
		ELSIF Azs.bError THEN
			StepA.step := StepA.step + 10000;
		END_IF
		
	235:
		tmr01A.IN := TRUE;
		tmr01A.PT := T#2S;
		IF tmr01A.Q THEN
			tmr01A.IN := FALSE;
			StepA.step := StepA.step + 1;
		END_IF
		
	236:
		StepA.step := 240;
		
		
	240:
		moveZdis := DisSensor_Dis - Macfg.laserA_Dis;
		StepA.step := StepA.step + 1;
		
	241:
		Az.RelMove(moveZdis * -1, SpdC.LowSpeed);
		StepA.step := StepA.step + 1;
		
	242:
		IF Azs.bBuzy OR Azs.bError THEN
			StepA.step := StepA.step + 1;
		END_IF
		
	243:
		IF Azs.bDone THEN
			StepA.step := StepA.step + 1;
		ELSIF Azs.bError THEN
			StepA.step := StepA.step + 10000;
		END_IF
		
	244:
		StepA.step := 250;
		
	250:
		z_PosMeasure := GaZ.Pos;
		StepA.bDone := TRUE;
		StepA.step	:= 0;
		
END_CASE
END_ACTION

ACTION Step_A_03_FindY:
CASE StepA.step OF
	300: // 判斷當距離再200~400間，才做偵測
		IF DisSensor_Dis > 200 OR DisSensor_Dis < 400 THEN
			StepA.step := StepA.step + 1;
		ELSE
			pmsg.Push_Alarm_NoPause("GroupA:Z軸距離感應器不再感應範圍內，取消Y軸原點偵測，使用預設值");
			StepA.step	:= 380;
		END_IF
		
	301:
		StepA.step := 310;
		
	310: 
		Ay.AbsMove(100, 50);
		StepA.step := StepA.step + 1;
		
	311:
		IF Ays.bBuzy OR Ays.bError THEN
			StepA.step := StepA.step + 1;
		END_IF
		
	312:
		IF NOT DisSensor_SSC1 THEN
			Ay.Stop();
			StepA.step := StepA.step + 1;
		ELSIF Ays.bDone THEN
			pmsg.Push_Alarm_NoPause("GroupA:Z軸距離感應器訊號錯誤");
			StepA.step := 380;
		ELSIF Ays.bError THEN
			StepA.step := StepA.step + 10000;
		END_IF
		
	313:
		tmr01A.IN := TRUE;
		tmr01A.PT := T#500MS;
		IF tmr01A.Q THEN
			tmr01A.IN := FALSE;
			StepA.step := StepA.step + 1;
		END_IF
		
	314:
		StepA.step := 320;
		
	320:
		Ay.AbsMove(Ay_P_Limite - 5, 5);
		StepA.step := StepA.step + 1;
		
	321:
		IF (Ays.bBuzy OR Ays.bError) THEN
			StepA.step := StepA.step + 1;
		END_IF
		
	322:
		IF DisSensor_SSC1 THEN
			Ay.Stop();
			StepA.step := StepA.step + 1;
		ELSIF Ays.bDone THEN
			pmsg.Push_Alarm_NoPause("GroupA:Z軸距離感應器訊號錯誤");
			StepA.step := 380;
		ELSIF Ays.bError THEN
			StepA.step := StepA.step + 10000;
		END_IF
		
	323:
		tmr01A.IN := TRUE;
		tmr01A.PT := T#500MS;
		IF tmr01A.Q THEN
			tmr01A.IN := FALSE;
			StepA.step := StepA.step + 1;
		END_IF
		
	324:
		StepA.step := 330;
		
		
	330:
		Ay.AbsMove(100, 0.5);
		StepA.step := StepA.step + 1;
		
	331:
		IF Ays.bBuzy OR Ays.bError THEN
			StepA.step := StepA.step + 1;
		END_IF
		
	332:
		IF NOT DisSensor_SSC1 THEN
			Ay.Stop();
			StepA.step := StepA.step + 1;
		ELSIF Ays.bDone THEN
			pmsg.Push_Alarm_NoPause("GroupA:Z軸距離感應器訊號錯誤");
			StepA.step := 380;
		ELSIF Ays.bError THEN
			StepA.step := StepA.step + 10000;
		END_IF
		
	333:
		tmr01A.IN := TRUE;
		tmr01A.PT := T#500MS;
		IF tmr01A.Q THEN
			tmr01A.IN := FALSE;
			StepA.step := StepA.step + 1;
		END_IF
		
	334:
		StepA.step := 340;
		
		
	340:
		Set_Y_Ref(Ay.Pos);
		StepA.step := StepA.step + 1;
		
	341:
		StepA.step := 390;
		
	
	380:
		IF projectData.Now_Steel.Width > 0 THEN
			Set_Y_Ref(Ay_P_Limite + 56 - projectData.Now_Steel.Width);
		ELSE
			Set_Y_Ref(Ay_P_Limite + 56 - 500);
		END_IF
		StepA.step := StepA.step + 1;
		
	381:
		StepA.step	:= 390;
	
	390:
		z_PosMeasure := GaZ.Pos;
		StepA.bDone := TRUE;
		StepA.step	:= 0;
		
END_CASE
END_ACTION

ACTION Step_A_10_MoveToXY_REF:
CASE StepA.step OF
	1000:// 計算相對距離
		tmpPos_X := moveCmd_X - pointRef.X;
		tmpPos_Y := moveCmd_Y + pointRef.Y;
		Dxf_Y_Move := 0;
		StepA.step := StepA.step + 1;
		
	1001:
		IF tmpPos_X < Ax_P_Limite AND tmpPos_X > Ax_N_Limite THEN
			StepA.step := StepA.step + 1;
		ELSIF tmpPos_X >= Ax_P_Limite THEN
			StepA.step := StepA.step + 10000;
			pMsg.Push_Alarm("GroupA MoveXY:命令位置超出X軸+極限");
		ELSE
			StepA.step := StepA.step + 10000;
			pMsg.Push_Alarm("GroupA MoveXY:命令位置超出X軸-極限");
		END_IF
 
			
	1002:
		IF tmpPos_Y < Ay_P_Limite - 5 AND tmpPos_Y > Ay_N_Limite THEN
			StepA.step := StepA.step + 1;
		ELSIF tmpPos_Y >= Ay_P_Limite - 5 THEN
			Dxf_Y_Move := tmpPos_Y - (Ay_P_Limite - 5);
			IF Dxf_Y_Move >= 70 THEN 
				StepA.step := StepA.step + 10000;
				pMsg.Push_Alarm("GroupA MoveXY_Ref:命令位置超出Y軸+極限");
			ELSE
				tmpPos_Y := (Ay_P_Limite - 5);
				StepA.step := StepA.step + 1;
			END_IF
		ELSE
			StepA.step := StepA.step + 10000;
			pMsg.Push_Alarm("GroupA MoveXY_Ref:命令位置超出Y軸-極限");
		END_IF
		
	1003:
		StepA.step := 1010;
		
	1010:
		Ax.AbsMove(tmpPos_X, moveCmd_Spd);
		Ay.AbsMove(tmpPos_Y, moveCmd_Spd);
		StepA.step := StepA.step + 1;
		
	1011:
		IF (Axs.bBuzy OR Axs.bError) AND (Ays.bBuzy OR Ays.bError) THEN
			StepA.step := StepA.step + 1;
		END_IF
		
	1012:
		IF Axs.bDone AND Ays.bDone THEN
			StepA.step := StepA.step + 1;
		ELSIF Axs.bError OR Ays.bError THEN
			StepA.step := StepA.step + 10000;
		END_IF
		
	1013:
		tmr01A.IN := TRUE;
		tmr01A.PT := T#1S;
		IF tmr01A.Q THEN
			tmr01A.IN := FALSE;
			StepA.step := StepA.step + 1;
		END_IF
		
	1014:
		StepA.step := 1020;
		
	1020:
		StepA.bDone := TRUE;
		StepA.step := 0;
		
END_CASE
END_ACTION

ACTION Step_A_20_ToStanbyPos:


CASE StepA.step OF
	2000:
		StepA.step := 2010;
		
	2010:
		IF GaZ.Pos > posc.pos_GaZ_stanby - 20 THEN
			StepA.step := 2020;
		ELSE
			StepA.step := StepA.step + 1;
		END_IF
		
	2011:
		Az.RelMove(20, moveCmd_Spd);
		StepA.step := StepA.step + 1;
		
	2012:
		IF Azs.bDone OR Azs.bError THEN
			StepA.step := StepA.step + 1;
		END_IF
		
	2013:
		IF Azs.bDone THEN
			StepA.step := StepA.step + 1;
		ELSIF Azs.bError THEN
			StepA.step := StepA.step + 10000;
		END_IF
		
	2014:
		StepA.step := 2020;
		
	2020:
		Ax.AbsMove(posc.pos_GaX_stanby, moveCmd_Spd);
		StepA.step := StepA.step + 1;
		
	2021:
		IF (Axs.bBuzy OR Axs.bError) THEN
			StepA.step := StepA.step + 1;
		END_IF
		
	2022:
		IF Axs.bDone THEN
			StepA.step := StepA.step + 1;
		ELSIF Axs.bError THEN
			StepA.step := StepA.step + 10000;
		END_IF
	
	2023:
		StepA.step := 2030;
	
	2030:
		GaZ.AbsMove(posc.pos_GaZ_stanby, moveCmd_Spd);
		GaY.AbsMove(posc.pos_GaY_stanby, moveCmd_Spd);
		StepA.step := StepA.step + 1;
		
	2031:
		IF (Azs.bBuzy OR Azs.bError) AND (Ays.bBuzy OR Ays.bError)  THEN
			StepA.step := StepA.step + 1;
		END_IF
		
	2032:
		IF Azs.bDone AND Ays.bDone THEN
			StepA.step := StepA.step + 1;
		ELSIF Azs.bError OR Ays.bError THEN
			StepA.step := StepA.step + 10000;
		END_IF
		
	2033:
		StepA.step := 2040;
		
		
	2040:
		StepA.bDone := TRUE;
		StepA.step := 0;
		
END_CASE
END_ACTION

ACTION Timer:
tmr01A();
tmr01();
tmr02();

// tmr_oil(in := IO.q204 AND IO.i302, PT:=T#2S);
tmr_oil(in := IO.q204 , PT:=T#2S);



IF tmr_oil.Q THEN
	IO.q204 := FALSE;
	
	Axis.GaX_Last_Oil := Axis.GaX_total_Move;
	
	Axis.GaY_Last_Oil := Axis.GaY_total_Move;
	
	Axis.GaZ_Last_Oil := Axis.GaZ_total_Move;
END_IF
END_ACTION

METHOD ToStanby : BOOL
VAR_INPUT
	Speed : LREAL := 0;
END_VAR
StepA.bDone := FALSE;
IF Speed > 0 THEN
	moveCmd_Spd := Speed;
ELSE
	moveCmd_Spd := SpdC.HomeSpeed;
END_IF

// ============ 紀錄啟動條件 ============
_logA.fbJson.StartObject();
_logA.fbJson.AddKeyString('MethodName','ToStanby');
_logA.fbJson.AddKeyLreal('Velocity', Speed);
_logA.JsonOutput();
// ======================================


StepA.step := 2000;
END_METHOD

METHOD XY_Move : BOOL
VAR_INPUT
	X_Point : REAL;
	Y_Point	: REAL;
	Speed : REAL;
END_VAR
moveCmd_X := X_Point;
moveCmd_Y := Y_Point;
moveCmd_Spd := Speed;

StepA.bDone := FALSE;

// ============ 紀錄啟動條件 ============
_logA.fbJson.StartObject();
_logA.fbJson.AddKeyString('MethodName','XY_Move');
_logA.fbJson.AddKeyLreal('X_Point', X_Point);
_logA.fbJson.AddKeyLreal('Y_Point', Y_Point);
_logA.fbJson.AddKeyLreal('Velocity', Speed);
_logA.JsonOutput();
// ======================================


StepA.step := 100;
END_METHOD

METHOD XY_Move_Ref : BOOL
VAR_INPUT
	X_Point : LREAL;
	Y_Point	: LREAL;
	Speed : LREAL;
END_VAR
moveCmd_X := X_Point;
moveCmd_Y := Y_Point;
moveCmd_Spd := Speed;

StepA.bDone := FALSE;

// ============ 紀錄啟動條件 ============
_logA.fbJson.StartObject();
_logA.fbJson.AddKeyString('MethodName','XY_Move_Ref');
_logA.fbJson.AddKeyLreal('X_Point', X_Point);
_logA.fbJson.AddKeyLreal('Y_Point', Y_Point);
_logA.fbJson.AddKeyLreal('Velocity', Speed);
_logA.JsonOutput();
// ======================================


StepA.step := 1000;
END_METHOD

END_PROGRAM

// ---- POUs/硬體控制/測距感應器/Sensor.TcPOU
PROGRAM Sensor
VAR
	sensorA	: OMH555_Decoder;
	sensorB : OMH555_Decoder;
	sensorC : OMH555_Decoder;
	sensorD : OMH555_Decoder;
	
	sensor_test_pos : LREAL;
	
	Sensor_Maintenance_required : ARRAY [0..3] OF BOOL;

END_VAR

VAR_INPUT
	Set_SensoeZero: BOOL;
END_VAR

// 測距感應器
sensorA();
sensorB();
sensorc();
sensorD();


IF Sensor_Maintenance_required[0] <> sensorA.bMaintenance_required THEN
	IF sensorA.bMaintenance_required THEN
		pMsg.Push_Alarm("雷射頭A: 測距感應器需要維護");
	END_IF
	Sensor_Maintenance_required[0] := sensorA.bMaintenance_required;
END_IF

IF Sensor_Maintenance_required[1] <> sensorB.bMaintenance_required THEN
	IF sensorB.bMaintenance_required THEN
		pMsg.Push_Alarm("雷射頭B: 測距感應器需要維護");
	END_IF
	Sensor_Maintenance_required[1] := sensorB.bMaintenance_required;
END_IF

IF Sensor_Maintenance_required[2] <> sensorC.bMaintenance_required THEN
	IF sensorC.bMaintenance_required THEN
		pMsg.Push_Alarm("雷射頭C: 測距感應器需要維護");
	END_IF
	Sensor_Maintenance_required[2] := sensorC.bMaintenance_required;
END_IF

IF Sensor_Maintenance_required[3] <> sensorD.bMaintenance_required THEN
	IF sensorD.bMaintenance_required THEN
		pMsg.Push_Alarm("雷射頭D: 測距感應器需要維護");
	END_IF
	Sensor_Maintenance_required[3] := sensorD.bMaintenance_required;
END_IF

END_PROGRAM

// ---- POUs/硬體控制/測距感應器/OMH555_Decoder.TcPOU
FUNCTION_BLOCK OMH555_Decoder IMPLEMENTS I_DisSensor
VAR_INPUT
END_VAR
VAR_OUTPUT
	// 距離 (單位:mm)
	fDistance : REAL;
	// 裝置狀態正常
	SSC1_1			:BOOL;
	// 裝置狀態正常
	bDevice_is_OK			:BOOL;
	// 需要維護
	bMaintenance_required	:BOOL;
	// 超出測量距離
	bOut_of_specification	:BOOL;
	// 檢查功能
	bFunctional_check		:BOOL;
	// 錯誤
	bFailure				:BOOL;
	// 距離比例(單位:公尺)
	iScale_Distance			:INT;
END_VAR
VAR
	// 原始資料輸入
	in_RawData AT %I* : ARRAY [0..3] OF USINT;
	// 原始資料輸出
	out_rawdata AT %Q* :USINT;	
	
	

	DistanceTmp : DINT;
	tmpStatus : WORD;
	tmpStatus2 : WORD;
	tmpStatus3 : DWORD;
	tmpfDistance : POINTER TO SINT;
END_VAR

DistanceTmp := (in_RawData[0] * 16#FF) +  (in_RawData[1] -10 );
tmpfDistance := ADR(in_RawData[2]);


IF (DistanceTmp >= 500) AND (DistanceTmp <= 5000) THEN
	fDistance := DINT_TO_REAL(DistanceTmp) * 0.1;
ELSE
	fDistance := 0;
END_IF

tmpStatus := ROR(in_RawData[3] AND 16#F0, 4);

SSC1_1 := (in_RawData[3] AND 16#1) = 1;

bDevice_is_OK := tmpStatus = 0;
bMaintenance_required := tmpStatus = 1;
bOut_of_specification := tmpStatus = 2;
bFunctional_check := tmpStatus = 3;
bFailure := tmpStatus = 4;

tmpStatus2 := 0;

out_rawdata := WORD_TO_USINT(tmpStatus2);

PROPERTY Distance : LREAL
GET
Distance := fDistance;
END_GET
END_PROPERTY

END_FUNCTION_BLOCK

// ---- POUs/功能塊/資料庫 Postgre相關/ReadSQLData.TcPOU
PROGRAM ReadSQLData
VAR
	step : INT;	

	_fb_PLCDBCmdEvt : FB_PLCDBCmdEvt(sNetID:= '', tTimeout:= T#5S );
	
	_SqlCommand : STRING(1024);
	
	// 讀回的資料筆數
	read_num: UDINT;
	
	// 帶入參數
	_stPara		: ARRAY [0..5] OF ST_ExpParameter;
	
	tcMessage     : I_TcMessage;
	
	database_server_id: UDINT := 2;
	
	_uuid : STRING(36);
	
	// 取得加工起始點的 SQL資料查詢結構
	_GetPosX : SQL_GetPosX_Struct;
	
	// 取得加工資料 的 資料查詢結構
	_Get_Payload : SQL_Get_Payload_Struct;
	
	_DataExists :BOOL;
	
	// 使用暫存器
	_FileBuffNumber	: INT;
	
	
	// 寫入啟動時間
	Write_Time_para : Payload_Write_Time;
	
	
	// 使用雷射參數
	_ParaNum : INT;
	
	// 使用暫存器
	_ParaBuffNumber	: INT;
	
	_fb_FileOpen : FB_FileOpen ;
	
	_e_OpenPath : E_OpenPath;
	
	_fb_FileWrite : FB_FileWrite;
	
	_fb_FileClose : FB_FileClose;
	
	test: PVOID;
	TmrWdt: TON;
	
	systime         : FB_LocalSystemTime;
	currentTime     : DT;
	
	_sn_cnt1 : UDINT;
END_VAR

VAR_OUTPUT
	bBuzy	: BOOL;
	bDone	: UDINT;
	bError	: BOOL;
	
	fNext_XPos	: LREAL;
	
	stLaserParameter : LaserParameter_Data;
END_VAR


bBuzy := step > 0 AND step < 10000;

bError := step > 10000;

IF bBuzy OR bError THEN
	bDone := 0;
END_IF

TmrWdt(in := bBuzy, PT:=T#20S);
IF TmrWdt.Q THEN
	pMsg.Push_Alarm_NoPause(
				WStrConcat("ReadSQLData", ":功能執行超時", TO_WSTRING(step))
			);
	step := step + 10000;
END_IF

IF step = 0 THEN
	RETURN;
END_IF

systime(
	bEnable:= TRUE, 
	dwCycle:= 1,
	systemTime=> );
currentTime := SYSTEMTIME_TO_DT(systime.systemTime);

Stap_0100_Get_Work_Order();
	
Stap_0200_Get_SteelData_X();

Stap_0300_Get_Payload_DataNum();

Stap_0400_Get_Payload_Data();

Stap_0500_Get_X_Next_StartPos();

Stap_1200_Get_Steel_Num_On_Wait();

Stap_2000_Set_Payload_Start();

Stap_2100_Set_Payload_Finish();

Stap_3000_Set_Steel_Start();

Stap_3100_Set_Steel_Finish();

Stap_3200_Set_Steel_SN();

METHOD Get_DxfFile : UDINT
VAR_INPUT
	// 檔案的UUID
	dataUuid : STRING(36);
	
	// 使用DXF檔案暫存
	BufferNumber : int;
END_VAR

IF NOT bBuzy THEN
	_uuid := dataUuid;
	
	_FileBuffNumber := BufferNumber;
	
	bdone := 0;
	
	bBuzy := TRUE;
	
	step := 1000;
	
	_sn_cnt1 := _sn_cnt1 + 1;
	
	Get_DxfFile := _sn_cnt1;
ELSE
	Get_DxfFile := 0;
END_IF
END_METHOD

METHOD Get_LaserParame : UDINT
VAR_INPUT
	// 讀取的參數ID
	paramNum : INT;
	// 放到暫存區位置
	PutToMem :INT;
END_VAR
IF NOT bBuzy THEN
	_ParaNum := paramNum;
	
	_ParaBuffNumber := PutToMem;
	
	bdone := 0;
	
	bBuzy := TRUE;
	
	step := 600;
	
	_sn_cnt1 := _sn_cnt1 + 1;
	
	Get_LaserParame := _sn_cnt1;
ELSE
	Get_LaserParame := 0;
END_IF
END_METHOD

METHOD Get_Payload : udint
VAR_INPUT
	// 區間的起始位置
	Start_Pos : LREAL;
	// 區間的結束位置
	End_Pos : LREAL;
END_VAR

// _Get_Payload.PosBegain := Start_Pos;
// _Get_Payload.PosEnd := End_Pos;
// 
// bdone := FALSE;
// 
// step := 300;
	
IF NOT bBuzy THEN
	_Get_Payload.PosBegain := Start_Pos;
	_Get_Payload.PosEnd := End_Pos;
	
	bdone := 0;
	
	bBuzy := TRUE;
	
	step := 300;
	
	_sn_cnt1 := _sn_cnt1 + 1;
	
	Get_Payload := _sn_cnt1;
ELSE
	Get_Payload := 0;
END_IF
END_METHOD

METHOD Get_Steel_Num_On_Wait : udint
VAR_INPUT
END_VAR
IF NOT bBuzy THEN
	bdone := 0;
	
	bBuzy := TRUE;
	
	step := 1200;
	
	_sn_cnt1 := _sn_cnt1 + 1;
	
	Get_Steel_Num_On_Wait := _sn_cnt1;
ELSE
	Get_Steel_Num_On_Wait := 0;
END_IF
END_METHOD

METHOD Get_SteelData : udint
VAR_INPUT
	UUID : STRING;
END_VAR
// _uuid := UUID;
// 
// bdone := FALSE;
// 
// step := 200;

IF NOT bBuzy THEN
	_uuid := UUID;
	
	bdone := 0;
	
	bBuzy := TRUE;
	
	step := 200;
	
	_sn_cnt1 := _sn_cnt1 + 1;
	
	Get_SteelData := _sn_cnt1;
ELSE
	Get_SteelData := 0;
END_IF
END_METHOD

METHOD Get_WorkkOrder : udint
VAR_INPUT
END_VAR
IF NOT bBuzy THEN
	
	bdone := 0;
	
	bBuzy := TRUE;
	
	step := 100;
	
	_sn_cnt1 := _sn_cnt1 + 1;
	
	Get_WorkkOrder := _sn_cnt1;
ELSE
	Get_WorkkOrder := 0;
END_IF
END_METHOD

METHOD Get_X_NextPos : udint
VAR_INPUT
	Pos : LREAL;
END_VAR
IF NOT bBuzy THEN
	_GetPosX.Pos := Pos;
	
	bdone := 0;
	
	bBuzy := TRUE;
	
	step := 500;
	
	_sn_cnt1 := _sn_cnt1 + 1;
	
	Get_X_NextPos := _sn_cnt1;
ELSE
	Get_X_NextPos := 0;
END_IF
END_METHOD

METHOD Set_Payload_Finish : udint
VAR_INPUT
	uid : STRING(36);
END_VAR
IF NOT bBuzy THEN
	_uuid := uid;
	
	bdone := 0;
	
	bBuzy := TRUE;
	
	step := 2100;
	
	_sn_cnt1 := _sn_cnt1 + 1;
	
	Set_Payload_Finish := _sn_cnt1;
ELSE
	Set_Payload_Finish := 0;
END_IF
END_METHOD

METHOD Set_Payload_Start : udint
VAR_INPUT
	uid : STRING(36);
END_VAR
IF NOT bBuzy THEN
	_uuid := uid;
	
	bdone := 0;
	
	bBuzy := TRUE;
	
	step := 2000;
	
	_sn_cnt1 := _sn_cnt1 + 1;
	
	Set_Payload_Start := _sn_cnt1;
ELSE
	Set_Payload_Start := 0;
END_IF
END_METHOD

METHOD Set_Steel_Finish : udint
VAR_INPUT
	uid : STRING(36);
END_VAR
IF NOT bBuzy THEN
	_uuid := uid;
	
	bdone := 0;
	
	bBuzy := TRUE;
	
	step := 3100;
	
	_sn_cnt1 := _sn_cnt1 + 1;
	
	Set_Steel_Finish := _sn_cnt1;
ELSE
	Set_Steel_Finish := 0;
END_IF
END_METHOD

METHOD Set_Steel_Start : udint
VAR_INPUT
	uid : STRING(36);
END_VAR
IF NOT bBuzy THEN
	_uuid := uid;
	
	bdone := 0;
	
	bBuzy := TRUE;
	
	step := 3000;
	
	_sn_cnt1 := _sn_cnt1 + 1;
	
	Set_Steel_Start := _sn_cnt1;
ELSE
	Set_Steel_Start := 0;
END_IF
END_METHOD

ACTION Stap_0100_Get_Work_Order:
CASE step OF
	
	100:
		ProjectData.WorkOrder_inSide.SN := 0;
		ProjectData.WorkOrder_inSide.steel_id := ''; 
		ProjectData.WorkOrder_inSide.Width := 0; 
		ProjectData.WorkOrder_inSide.Height := 0; 
		step := step + 1;
		
	101:
		ProjectData.WorkOrder_alignment.SN := 0;
		ProjectData.WorkOrder_alignment.steel_id := ''; 
		ProjectData.WorkOrder_alignment.Width := 0; 
		ProjectData.WorkOrder_alignment.Height := 0; 
		step := step + 1;
		
	102:
		ProjectData.WorkOrder_inserts.SN := 0;
		ProjectData.WorkOrder_inserts.steel_id := ''; 
		ProjectData.WorkOrder_inserts.Width := 0; 
		ProjectData.WorkOrder_inserts.Height := 0; 
		step := step + 1;
		
	103:
		step := 110;

(*	===========================================
				抓取　inSide(入料)　資料
	===========================================*)	
	110:
		// SQL命令
		_SqlCommand := 
		'
		SELECT 
			"sequence_number", 
			s.height, 
			s.width, 
			CAST("part_nest_id" as char(36))
		FROM 
			"public"."work_order_data" 
		LEFT JOIN 
			"public"."steeldata" s 
		ON 
			s.id = part_nest_id::uuid
		WHERE
 			"steel_status" = $'inSide$'
		ORDER BY 
			"sequence_number"
		';

		
//		'SELECT  FROM dxf_data WHERE id = {id}::UUID';
	
		// 設定對應參數
		_stPara[0].sParaName := 'id'; 			_stPara[0].eParaType := E_ExpParameterType.STRING_; 		_stPara[0].nParaSize := SIZEOF(_uuid);
		step := step + 1;
		
	111:
		IF 
			MsgMain._fb_PLCDBCmdEvt.ExecuteDataReturn(
				hDBID := database_server_id,
				pExpression := ADR(_SqlCommand),			// SQL 命令 ex. SELECT * FROM PlcTest.newtable WHERE ID = {ID}  
				cbExpression := SIZEOF(_SqlCommand),		// SQL 命令字串的長度
				pData:= ADR(_uuid),							// 帶入的參數值
				cbData:= SIZEOF(_uuid),						// 帶入的參數值大小
				pParameter:= ADR(_stPara), 					// 帶入的參數類型設定  ex.上面命令內的 {ID} 類型設定
				cbParameter:= SIZEOF(_stPara[0]) * 1,		// 帶入的參數類型設定的大小
				nStartIndex := 0,
				nRecordCount := 32,
				pReturnData := ADR(ProjectData.WorkOrder_inSide),
				cbReturnData := SIZEOF(ProjectData.WorkOrder_inSide),
				pRecords := ADR(read_num)
			) 
		THEN
			IF MsgMain._fb_PLCDBCmdEvt.bError THEN
				tcMessage := MsgMain._fb_PLCDBCmdEvt.ipTcResult;
				step := step + 10000;
			ELSE
				step := step + 1;
			END_IF
			
		END_IF
		
	112:
		step := 120;

(*	===========================================
				抓取　inserts(差單) 與 continue(續接)　資料
	===========================================*)	
	120:
		// SQL命令
		_SqlCommand := 
		'
		SELECT 
			"sequence_number", 
			s.height, 
			s.width, 
			CAST("part_nest_id" as char(36))
		FROM 
			"public"."work_order_data" 
		LEFT JOIN 
			"public"."steeldata" s 
		ON 
			s.id = part_nest_id::uuid
		WHERE
 			"steel_status" = $'inserts$' OR "steel_status" = $'continue$'
		ORDER BY 
			"sequence_number"
		';

		
//		'SELECT  FROM dxf_data WHERE id = {id}::UUID';
	
		// 設定對應參數
		_stPara[0].sParaName := 'id'; 			_stPara[0].eParaType := E_ExpParameterType.STRING_; 		_stPara[0].nParaSize := SIZEOF(_uuid);
		step := step + 1;
		
	121:
		IF 
			MsgMain._fb_PLCDBCmdEvt.ExecuteDataReturn(
				hDBID := database_server_id,
				pExpression := ADR(_SqlCommand),			// SQL 命令 ex. SELECT * FROM PlcTest.newtable WHERE ID = {ID}  
				cbExpression := SIZEOF(_SqlCommand),		// SQL 命令字串的長度
				pData:= ADR(_uuid),							// 帶入的參數值
				cbData:= SIZEOF(_uuid),						// 帶入的參數值大小
				pParameter:= ADR(_stPara), 					// 帶入的參數類型設定  ex.上面命令內的 {ID} 類型設定
				cbParameter:= SIZEOF(_stPara[0]) * 0,		// 帶入的參數類型設定的大小
				nStartIndex := 0,
				nRecordCount := 32,
				pReturnData := ADR(ProjectData.WorkOrder_inserts),
				cbReturnData := SIZEOF(ProjectData.WorkOrder_inserts),
				pRecords := ADR(read_num)
			) 
		THEN
			IF MsgMain._fb_PLCDBCmdEvt.bError THEN
				tcMessage := MsgMain._fb_PLCDBCmdEvt.ipTcResult;
				step := step + 10000;
			ELSE
				step := step + 1;
			END_IF
			
		END_IF
		
	122:
		step := 130;
		
(*	===========================================
				抓取無靠邊差單資料
	===========================================*)		
		
	130:
		// SQL命令
		_SqlCommand := 
		'
		SELECT 
			"sequence_number", 
			s.height, 
			s.width, 
			CAST("part_nest_id" as char(36))
		FROM 
			"public"."work_order_data" 
		LEFT JOIN 
			"public"."steeldata" s 
		ON 
			s.id = part_nest_id::uuid
		WHERE
 			"steel_status" = $'alignment$'
		ORDER BY 
			"sequence_number"
		';

		
//		'SELECT  FROM dxf_data WHERE id = {id}::UUID';
	
		// 設定對應參數
		_stPara[0].sParaName := 'id'; 			_stPara[0].eParaType := E_ExpParameterType.STRING_; 		_stPara[0].nParaSize := SIZEOF(_uuid);
		step := step + 1;
		
	131:
		IF 
			MsgMain._fb_PLCDBCmdEvt.ExecuteDataReturn(
				hDBID := database_server_id,
				pExpression := ADR(_SqlCommand),			// SQL 命令 ex. SELECT * FROM PlcTest.newtable WHERE ID = {ID}  
				cbExpression := SIZEOF(_SqlCommand),		// SQL 命令字串的長度
				pData:= ADR(_uuid),							// 帶入的參數值
				cbData:= SIZEOF(_uuid),						// 帶入的參數值大小
				pParameter:= ADR(_stPara), 					// 帶入的參數類型設定  ex.上面命令內的 {ID} 類型設定
				cbParameter:= SIZEOF(_stPara[0]) * 0,		// 帶入的參數類型設定的大小
				nStartIndex := 0,
				nRecordCount := 32,
				pReturnData := ADR(ProjectData.WorkOrder_alignment),
				cbReturnData := SIZEOF(ProjectData.WorkOrder_alignment),
				pRecords := ADR(read_num)
			) 
		THEN
			IF MsgMain._fb_PLCDBCmdEvt.bError THEN
				tcMessage := MsgMain._fb_PLCDBCmdEvt.ipTcResult;
				step := step + 10000;
			ELSE
				step := step + 1;
			END_IF
			
		END_IF
		
	132:
		bDone := _sn_cnt1;
		step := 0;
END_CASE
END_ACTION

ACTION Stap_0200_Get_SteelData_X:
CASE step OF
	200:
		step := step + 1;

	201:
		// SQL命令
		_SqlCommand := 
		'SELECT 
			CAST("id" as char(36)),
			"steeltype", 
			"length", 
			"height", 
			"width", 
			"t1", 
			"t2", 
			"origin_offset", 
			"preview_enabled", 
			"preview_mode", 
			"preview_tme", 
			"designate_area_range_begin", 
			"designate_area_range_end", 
			CAST("payloadtop" as char(36)), 
			CAST("payloadbottom" as char(36)), 
			CAST("payloadleft" as char(36)), 
			CAST("payloadright" as char(36)), 
			"is_job_finish"
		FROM 
			"public"."steeldata"
		WHERE
			"id" = {id}::UUID';
//		'SELECT  FROM dxf_data WHERE id = {id}::UUID';
	
		// 設定對應參數
		_stPara[0].sParaName := 'id'; 			_stPara[0].eParaType := E_ExpParameterType.STRING_; 		_stPara[0].nParaSize := SIZEOF(_uuid);
		step := step + 1;
		
	202:
		IF 
			MsgMain._fb_PLCDBCmdEvt.ExecuteDataReturn(
				hDBID := database_server_id,
				pExpression := ADR(_SqlCommand),			// SQL 命令 ex. SELECT * FROM PlcTest.newtable WHERE ID = {ID}  
				cbExpression := SIZEOF(_SqlCommand),		// SQL 命令字串的長度
				pData:= ADR(_uuid),							// 帶入的參數值
				cbData:= SIZEOF(_uuid),						// 帶入的參數值大小
				pParameter:= ADR(_stPara), 					// 帶入的參數類型設定  ex.上面命令內的 {ID} 類型設定
				cbParameter:= SIZEOF(_stPara[0]) * 1,		// 帶入的參數類型設定的大小
				nStartIndex := 0,
				nRecordCount := 1,
				pReturnData := ADR(ProjectData.Now_Steel),
				cbReturnData := SIZEOF(ProjectData.Now_Steel),
				pRecords := ADR(read_num)
			) 
		THEN
			IF MsgMain._fb_PLCDBCmdEvt.bError THEN
				tcMessage := MsgMain._fb_PLCDBCmdEvt.ipTcResult;
				step := step + 10000;
			ELSE
				step := step + 1;
			END_IF
			
		END_IF
		
	203:
		bDone := _sn_cnt1;
		step := 0;
END_CASE
END_ACTION

ACTION Stap_0300_Get_Payload_DataNum:
CASE step OF
	300:
		IF _Get_Payload.PosEnd <= _Get_Payload.PosBegain THEN
			_Get_Payload.PosEnd := _Get_Payload.PosBegain + 300;
		END_IF
		step := step + 1;
		
		
(*	===============================
		取得左面(Ga)的資料數量
	===============================	*)
	301: 
		_Get_Payload.Payload_Uid := ProjectData.Now_Steel.payloadLeft;
		// SQL命令
		_SqlCommand := 
		'SELECT
			Count(*)::int2
		FROM 
			payloaddata
		WHERE
			payload_uid = {id} AND
			"point_x" >= {PosBegain} AND
			"point_x" < {PosEnd} AND
			is_stage_finish = false
			';
	
		// 設定對應參數
		_stPara[0].sParaName := 'id'; 			_stPara[0].eParaType := E_ExpParameterType.STRING_; 		_stPara[0].nParaSize := 37;
		_stPara[1].sParaName := 'PosBegain'; 	_stPara[1].eParaType := E_ExpParameterType.Double64; 		_stPara[1].nParaSize := 8;
		_stPara[2].sParaName := 'PosEnd'; 		_stPara[2].eParaType := E_ExpParameterType.Double64; 		_stPara[2].nParaSize := 8;
		step := step + 1;
		
	302:
		IF 
			MsgMain._fb_PLCDBCmdEvt.ExecuteDataReturn(
				hDBID := database_server_id,
				pExpression := ADR(_SqlCommand),			// SQL 命令 ex. SELECT * FROM PlcTest.newtable WHERE ID = {ID}  
				cbExpression := SIZEOF(_SqlCommand),		// SQL 命令字串的長度
				pData:= ADR(_Get_Payload),							// 帶入的參數值
				cbData:= SIZEOF(_Get_Payload),						// 帶入的參數值大小
				pParameter:= ADR(_stPara), 					// 帶入的參數類型設定  ex.上面命令內的 {ID} 類型設定
				cbParameter:= SIZEOF(_stPara[0]) * 3,		// 帶入的參數類型設定的大小
				nStartIndex := 0,
				nRecordCount := 1,
				pReturnData := ADR(ProjectData.Now_Steel_Payload_A_DataNumber),
				cbReturnData := SIZEOF(ProjectData.Now_Steel_Payload_A_DataNumber),
				pRecords := ADR(read_num)
			) 
		THEN
			IF MsgMain._fb_PLCDBCmdEvt.bError THEN
				tcMessage := MsgMain._fb_PLCDBCmdEvt.ipTcResult;
				step := step + 10000;
			ELSE
				step := step + 1;
			END_IF
			
		END_IF
		
	303:
		step := 310;
		
(*	===============================
		取得上面(Gb)的資料數量
	===============================	*)
	310: // 取得此面的資料數量
		_Get_Payload.Payload_Uid := ProjectData.Now_Steel.payloadTop;
		step := step + 1;
		
	311:
		IF 
			MsgMain._fb_PLCDBCmdEvt.ExecuteDataReturn(
				hDBID := database_server_id,
				pExpression := ADR(_SqlCommand),			// SQL 命令 ex. SELECT * FROM PlcTest.newtable WHERE ID = {ID}  
				cbExpression := SIZEOF(_SqlCommand),		// SQL 命令字串的長度
				pData:= ADR(_Get_Payload),							// 帶入的參數值
				cbData:= SIZEOF(_Get_Payload),						// 帶入的參數值大小
				pParameter:= ADR(_stPara), 					// 帶入的參數類型設定  ex.上面命令內的 {ID} 類型設定
				cbParameter:= SIZEOF(_stPara[0]) * 3,		// 帶入的參數類型設定的大小
				nStartIndex := 0,
				nRecordCount := 1,
				pReturnData := ADR(ProjectData.Now_Steel_Payload_B_DataNumber),
				cbReturnData := SIZEOF(ProjectData.Now_Steel_Payload_B_DataNumber),
				pRecords := ADR(read_num)
			) 
		THEN
			IF MsgMain._fb_PLCDBCmdEvt.bError THEN
				tcMessage := MsgMain._fb_PLCDBCmdEvt.ipTcResult;
				step := step + 10000;
			ELSE
				step := step + 1;
			END_IF
			
		END_IF
		
	312:
		step := 320;
		
(*	===============================
		取得右面(Gc)的資料數量
	===============================	*)
	320: // 取得此面的資料數量
		_Get_Payload.Payload_Uid := ProjectData.Now_Steel.payloadRight;
		step := step + 1;
		
	321:
		IF 
			MsgMain._fb_PLCDBCmdEvt.ExecuteDataReturn(
				hDBID := database_server_id,
				pExpression := ADR(_SqlCommand),			// SQL 命令 ex. SELECT * FROM PlcTest.newtable WHERE ID = {ID}  
				cbExpression := SIZEOF(_SqlCommand),		// SQL 命令字串的長度
				pData:= ADR(_Get_Payload),							// 帶入的參數值
				cbData:= SIZEOF(_Get_Payload),						// 帶入的參數值大小
				pParameter:= ADR(_stPara), 					// 帶入的參數類型設定  ex.上面命令內的 {ID} 類型設定
				cbParameter:= SIZEOF(_stPara[0]) * 3,		// 帶入的參數類型設定的大小
				nStartIndex := 0,
				nRecordCount := 1,
				pReturnData := ADR(ProjectData.Now_Steel_Payload_C_DataNumber),
				cbReturnData := SIZEOF(ProjectData.Now_Steel_Payload_C_DataNumber),
				pRecords := ADR(read_num)
			) 
		THEN
			IF MsgMain._fb_PLCDBCmdEvt.bError THEN
				tcMessage := MsgMain._fb_PLCDBCmdEvt.ipTcResult;
				step := step + 10000;
			ELSE
				step := step + 1;
			END_IF
			
		END_IF
		
	322:
		step := 330;
		
(*	===============================
		取得底面(Gd)的資料數量
	===============================	*)
	330:
		_Get_Payload.Payload_Uid := ProjectData.Now_Steel.payloadBottom;
		step := step + 1;
		
	331:
		IF 
			MsgMain._fb_PLCDBCmdEvt.ExecuteDataReturn(
				hDBID := database_server_id,
				pExpression := ADR(_SqlCommand),			// SQL 命令 ex. SELECT * FROM PlcTest.newtable WHERE ID = {ID}  
				cbExpression := SIZEOF(_SqlCommand),		// SQL 命令字串的長度
				pData:= ADR(_Get_Payload),							// 帶入的參數值
				cbData:= SIZEOF(_Get_Payload),						// 帶入的參數值大小
				pParameter:= ADR(_stPara), 					// 帶入的參數類型設定  ex.上面命令內的 {ID} 類型設定
				cbParameter:= SIZEOF(_stPara[0]) * 3,		// 帶入的參數類型設定的大小
				nStartIndex := 0,
				nRecordCount := 1,
				pReturnData := ADR(ProjectData.Now_Steel_Payload_D_DataNumber),
				cbReturnData := SIZEOF(ProjectData.Now_Steel_Payload_D_DataNumber),
				pRecords := ADR(read_num)
			) 
		THEN
			IF MsgMain._fb_PLCDBCmdEvt.bError THEN
				tcMessage := MsgMain._fb_PLCDBCmdEvt.ipTcResult;
				step := step + 10000;
			ELSE
				step := step + 1;
			END_IF
			
		END_IF
		
	332:
		step := 340;
		
	340:
		step := 400;
		
END_CASE
END_ACTION

ACTION Stap_0400_Get_Payload_Data:
CASE step OF
	400:
		step := step + 1;
	
	401:
		// SQL命令
		_SqlCommand := 
		'SELECT
			CAST("data_uuid" as char(36)), 
			CAST("payload_uid" as char(36)), 
			"payload_serial", 
			0, 
			"point_x", 
			"point_y", 
			"width", 
			"height", 
			"is_qrcode",
			"is_stage_finish",
			CAST("qrcode_data" as char(100))
		FROM
			"public"."payloaddata"
		WHERE
			payload_uid = {id} AND
			"point_x" >= {PosBegain} AND "point_x" < {PosEnd} AND
			is_stage_finish = false
		ORDER BY
			"payload_serial"';
			
		// 設定對應參數
		_stPara[0].sParaName := 'id'; 			_stPara[0].eParaType := E_ExpParameterType.STRING_; 		_stPara[0].nParaSize := 37;
		_stPara[1].sParaName := 'PosBegain'; 	_stPara[1].eParaType := E_ExpParameterType.Double64; 		_stPara[1].nParaSize := 8;
		_stPara[2].sParaName := 'PosEnd'; 		_stPara[2].eParaType := E_ExpParameterType.Double64; 		_stPara[2].nParaSize := 8;
			
		step := step + 1;
		
	402:
		step := 410;

(*	===============================
		取得左側面(Ga)的資料
	===============================	*)
	410:
		IF ProjectData.Now_Steel_Payload_A_DataNumber > 0 THEN
			step := step + 1;
		ELSE
			step := step + 10;
		END_IF
	
	411: // SQL命令
		_Get_Payload.Payload_Uid := ProjectData.Now_Steel.payloadLeft;
		step := step + 1;
		
	412:
		IF 
		MsgMain._fb_PLCDBCmdEvt.ExecuteDataReturn(
			hDBID := database_server_id,
			pExpression := ADR(_SqlCommand),			// SQL 命令 ex. SELECT * FROM PlcTest.newtable WHERE ID = {ID}  
			cbExpression := SIZEOF(_SqlCommand),		// SQL 命令字串的長度
			pData:= ADR(_Get_Payload),							// 帶入的參數值
			cbData:= SIZEOF(_Get_Payload),						// 帶入的參數值大小
			pParameter:= ADR(_stPara), 					// 帶入的參數類型設定  ex.上面命令內的 {ID} 類型設定
			cbParameter:= SIZEOF(_stPara[0]) * 3,			// 帶入的參數類型設定的大小
			nStartIndex := 0,
			nRecordCount := 100,
			pReturnData := ADR(ProjectData.Payload_A_Data_buff),
			cbReturnData := SIZEOF(ProjectData.Payload_A_Data_buff),
			pRecords := ADR(read_num)
		)
		THEN
			IF MsgMain._fb_PLCDBCmdEvt.bError THEN
				tcMessage := MsgMain._fb_PLCDBCmdEvt.ipTcResult;
				step := step + 10000;
			ELSE
				step := step + 1;
			END_IF
		END_IF
		
	413:
		step := 420;
		
(*	===============================
		取得頂部面(Gb)的資料
	===============================	*)
	420:
		IF ProjectData.Now_Steel_Payload_B_DataNumber > 0 THEN
			step := step + 1;
		ELSE
			step := step + 10;
		END_IF
	
	421: // SQL命令
		_Get_Payload.Payload_Uid := ProjectData.Now_Steel.payloadTop;
		step := step + 1;
		
	422:
		IF 
		MsgMain._fb_PLCDBCmdEvt.ExecuteDataReturn(
			hDBID := database_server_id,
			pExpression := ADR(_SqlCommand),			// SQL 命令 ex. SELECT * FROM PlcTest.newtable WHERE ID = {ID}  
			cbExpression := SIZEOF(_SqlCommand),		// SQL 命令字串的長度
			pData:= ADR(_Get_Payload),							// 帶入的參數值
			cbData:= SIZEOF(_Get_Payload),						// 帶入的參數值大小
			pParameter:= ADR(_stPara), 					// 帶入的參數類型設定  ex.上面命令內的 {ID} 類型設定
			cbParameter:= SIZEOF(_stPara[0]) * 3,			// 帶入的參數類型設定的大小
			nStartIndex := 0,
			nRecordCount := 100,
			pReturnData := ADR(ProjectData.Payload_B_Data_buff),
			cbReturnData := SIZEOF(ProjectData.Payload_B_Data_buff),
			pRecords := ADR(read_num)
		)
		THEN
			IF MsgMain._fb_PLCDBCmdEvt.bError THEN
				tcMessage := MsgMain._fb_PLCDBCmdEvt.ipTcResult;
				step := step + 10000;
			ELSE
				step := step + 1;
			END_IF
		END_IF
		
	423:
		step := 430;
		
(*	===============================
		取得頂部面(Gc)的資料
	===============================	*)
	430:
		IF ProjectData.Now_Steel_Payload_C_DataNumber > 0 THEN
			step := step + 1;
		ELSE
			step := step + 10;
		END_IF
	
	431: // SQL命令
		_Get_Payload.Payload_Uid := ProjectData.Now_Steel.payloadRight;
		step := step + 1;
		
	432:
		IF 
		MsgMain._fb_PLCDBCmdEvt.ExecuteDataReturn(
			hDBID := database_server_id,
			pExpression := ADR(_SqlCommand),			// SQL 命令 ex. SELECT * FROM PlcTest.newtable WHERE ID = {ID}  
			cbExpression := SIZEOF(_SqlCommand),		// SQL 命令字串的長度
			pData:= ADR(_Get_Payload),							// 帶入的參數值
			cbData:= SIZEOF(_Get_Payload),						// 帶入的參數值大小
			pParameter:= ADR(_stPara), 					// 帶入的參數類型設定  ex.上面命令內的 {ID} 類型設定
			cbParameter:= SIZEOF(_stPara[0]) * 3,			// 帶入的參數類型設定的大小
			nStartIndex := 0,
			nRecordCount := 100,
			pReturnData := ADR(ProjectData.Payload_C_Data_buff),
			cbReturnData := SIZEOF(ProjectData.Payload_C_Data_buff),
			pRecords := ADR(read_num)
		)
		THEN
			IF MsgMain._fb_PLCDBCmdEvt.bError THEN
				tcMessage := MsgMain._fb_PLCDBCmdEvt.ipTcResult;
				step := step + 10000;
			ELSE
				step := step + 1;
			END_IF
		END_IF
		
	433:
		step := 440;
		
(*	===============================
		取得底部面(Gd)的資料
	===============================	*)
	440:
		IF ProjectData.Now_Steel_Payload_D_DataNumber > 0 THEN
			step := step + 1;
		ELSE
			step := step + 10;
		END_IF
	
	441: // SQL命令
		_Get_Payload.Payload_Uid := ProjectData.Now_Steel.payloadBottom;
		step := step + 1;
		
	442:
		IF 
		MsgMain._fb_PLCDBCmdEvt.ExecuteDataReturn(
			hDBID := database_server_id,
			pExpression := ADR(_SqlCommand),			// SQL 命令 ex. SELECT * FROM PlcTest.newtable WHERE ID = {ID}  
			cbExpression := SIZEOF(_SqlCommand),		// SQL 命令字串的長度
			pData:= ADR(_Get_Payload),							// 帶入的參數值
			cbData:= SIZEOF(_Get_Payload),						// 帶入的參數值大小
			pParameter:= ADR(_stPara), 									// 帶入的參數類型設定  ex.上面命令內的 {ID} 類型設定
			cbParameter:= SIZEOF(_stPara[0]) * 3,							// 帶入的參數類型設定的大小
			nStartIndex := 0,	// 起始的資料序號
			nRecordCount := 100,
			pReturnData := ADR(ProjectData.Payload_D_Data_buff),
			cbReturnData := SIZEOF(ProjectData.Payload_D_Data_buff),
			pRecords := ADR(read_num)
		)
		THEN
			IF MsgMain._fb_PLCDBCmdEvt.bError THEN
				tcMessage := MsgMain._fb_PLCDBCmdEvt.ipTcResult;
				step := step + 10000;
			ELSE
				step := step + 1;
			END_IF
		END_IF
		
	443:
		step := 450;
		
	450:
		bDone := _sn_cnt1;
		step := 0;
		
END_CASE
END_ACTION

ACTION Stap_0500_Get_X_Next_StartPos:
CASE step OF
 500:
		step := step + 1;
	
 501: 
		step := 510;

(*	===============================
		取得X最近點
	===============================	*)
 510:
		_GetPosX.Payload_A_Uid := ProjectData.Now_Steel.payloadTop;
		_GetPosX.Payload_B_Uid := ProjectData.Now_Steel.payloadBottom;
		_GetPosX.Payload_C_Uid := ProjectData.Now_Steel.payloadLeft;
		_GetPosX.Payload_D_Uid := ProjectData.Now_Steel.payloadRight;
		step := step + 1;
	
 511: // SQL命令
		_SqlCommand := 
		'SELECT
			"point_x"
		FROM
			"public"."payloaddata"
		WHERE
			(	
				"payload_uid" = {payload_uid_A} OR
				"payload_uid" = {payload_uid_B} OR 
				"payload_uid" = {payload_uid_C} OR 
				"payload_uid" = {payload_uid_D}
			) 
			AND
				is_stage_finish = false
			AND
				"point_x" > {PosX}
		ORDER BY
			"point_x"
		LIMIT 1';
	
		// 設定對應參數
		_stPara[0].sParaName := 'payload_uid_A';			_stPara[0].eParaType := E_ExpParameterType.STRING_;		_stPara[0].nParaSize := 37;
		_stPara[1].sParaName := 'payload_uid_B';			_stPara[1].eParaType := E_ExpParameterType.STRING_;		_stPara[1].nParaSize := 37;
		_stPara[2].sParaName := 'payload_uid_C';			_stPara[2].eParaType := E_ExpParameterType.STRING_;		_stPara[2].nParaSize := 37;
		_stPara[3].sParaName := 'payload_uid_D';			_stPara[3].eParaType := E_ExpParameterType.STRING_;		_stPara[3].nParaSize := 37;
		_stPara[4].sParaName := 'PosX';					_stPara[4].eParaType := E_ExpParameterType.Double64;	_stPara[4].nParaSize := 8;
		step := step + 1;
		
 512:
		IF 
		MsgMain._fb_PLCDBCmdEvt.ExecuteDataReturn(
			hDBID := database_server_id,
			pExpression := ADR(_SqlCommand),			// SQL 命令 ex. SELECT * FROM PlcTest.newtable WHERE ID = {ID}  
			cbExpression := SIZEOF(_SqlCommand),		// SQL 命令字串的長度
			pData:= ADR(_GetPosX),						// 帶入的參數值
			cbData:= SIZEOF(_GetPosX),					// 帶入的參數值大小
			pParameter:= ADR(_stPara), 					// 帶入的參數類型設定  ex.上面命令內的 {ID} 類型設定
			cbParameter:= SIZEOF(_stPara[0]) * 5,			// 帶入的參數類型設定的大小
			nStartIndex := 0,
			nRecordCount := 1,
			pReturnData := ADR(fNext_XPos),
			cbReturnData := SIZEOF(fNext_XPos),
			pRecords := ADR(read_num)
		)
		THEN
			IF MsgMain._fb_PLCDBCmdEvt.bError THEN
				tcMessage := MsgMain._fb_PLCDBCmdEvt.ipTcResult;
				step := step + 10000;
			ELSE
				IF read_num = 0 THEN
					fNext_XPos := -1;
				END_IF
				step := step + 1;
			END_IF
		END_IF
		
 513:
		bDone := _sn_cnt1;
		step := 0;
		
END_CASE
END_ACTION

ACTION Stap_1200_Get_Steel_Num_On_Wait:
CASE step OF
	
	1200:
		// SQL命令
		_SqlCommand := 
		'
		SELECT 
			Count(*)::int2
		FROM 
			"public"."work_order_data" 
		WHERE
 			"steel_status" = $'holding$' OR "steel_status" = $'waitLoading$'
		';

		step := step + 1;
		
	1201:
		IF 
			MsgMain._fb_PLCDBCmdEvt.ExecuteDataReturn(
				hDBID := database_server_id,
				pExpression := ADR(_SqlCommand),			// SQL 命令 ex. SELECT * FROM PlcTest.newtable WHERE ID = {ID}  
				cbExpression := SIZEOF(_SqlCommand),		// SQL 命令字串的長度
				pData:= 0,							// 帶入的參數值
				cbData:= 0,						// 帶入的參數值大小
				pParameter:= 0, 					// 帶入的參數類型設定  ex.上面命令內的 {ID} 類型設定
				cbParameter:= 0,		// 帶入的參數類型設定的大小
				nStartIndex := 0,
				nRecordCount := 1,
				pReturnData := ADR(ProjectData.WorkOrder_Num_On_Wait),
				cbReturnData := SIZEOF(ProjectData.WorkOrder_Num_On_Wait),
				pRecords := ADR(read_num)
			) 
		THEN
			IF MsgMain._fb_PLCDBCmdEvt.bError THEN
				tcMessage := MsgMain._fb_PLCDBCmdEvt.ipTcResult;
				step := step + 10000;
			ELSE
				step := step + 1;
			END_IF
			
		END_IF
		
	1202:
		bDone := _sn_cnt1;
		step := 0;
END_CASE
END_ACTION

ACTION Stap_2000_Set_Payload_Start:
(*	=================================================================
						從資料庫讀取 A頭 雷射檔
	================================================================= *)
CASE step OF
	2000:
		// SQL命令
		_SqlCommand := 
		'SELECT EXISTS(
			SELECT 
				data_uuid
			from 
				public.payloaddata
			where 
				data_uuid = {uuid}::uuid
		);';
		// 設定對應參數
		_stPara[0].sParaName := 'uuid'; 			_stPara[0].eParaType := E_ExpParameterType.STRING_; 		_stPara[0].nParaSize := 37;
		
		step := step + 1;
		
	2001:
		IF 
			MsgMain._fb_PLCDBCmdEvt.ExecuteDataReturn(
				hDBID := database_server_id,
				pExpression := ADR(_SqlCommand),			// SQL 命令 ex. SELECT * FROM PlcTest.newtable WHERE ID = {ID}  
				cbExpression := SIZEOF(_SqlCommand),		// SQL 命令字串的長度
				pData:= ADR(_uuid),							// 帶入的參數值
				cbData:= SIZEOF(_uuid),						// 帶入的參數值大小
				pParameter:= ADR(_stPara), 					// 帶入的參數類型設定  ex.上面命令內的 {ID} 類型設定
				cbParameter:= SIZEOF(_stPara[0]),		// 帶入的參數類型設定的大小
				nStartIndex := 0,
				nRecordCount := 1,
				pReturnData := ADR(_DataExists),
				cbReturnData := SIZEOF(_DataExists),
				pRecords := ADR(read_num)
			) 
		THEN
			IF MsgMain._fb_PLCDBCmdEvt.bError THEN
				tcMessage := MsgMain._fb_PLCDBCmdEvt.ipTcResult;
				step := step + 10000;
			ELSE
				step := step + 1;
			END_IF
			
		END_IF
		
	2002:
		IF _DataExists THEN
			step := step + 1;
		ELSE
			pmsg.Push_Alarm_NoPause(WStrConcat(str0:= "ReadSQLData.Set_Payload_Start: 讀取的UUID(", str1:= TO_WSTRING(_uuid), str2:= ")不存在。", str3:= TO_WSTRING(step)));
			step := step + 10000;
		END_IF
		
	2003:
			step := 2010;
			
	2010:
		Write_Time_para.Start_TIME := currentTime;
		Write_Time_para.Uid := _uuid;
	
		// SQL命令
		_SqlCommand := 
		'
		UPDATE 
			public.payloaddata 
		SET 
			stage_start = {timestamp}
		WHERE
			data_uuid = {id}::UUID
		';
		
	
		// 設定對應參數
		_stPara[0].sParaName := 'timestamp'; 			_stPara[0].eParaType := E_ExpParameterType.DateTime; 		_stPara[0].nParaSize := SIZEOF(Write_Time_para.Start_TIME);
		_stPara[1].sParaName := 'id'; 					_stPara[1].eParaType := E_ExpParameterType.STRING_; 		_stPara[1].nParaSize := 37;
		
		step := step + 1;
		
	2011:
		IF 
			MsgMain._fb_PLCDBCmdEvt.Execute(
				hDBID := database_server_id,
				pExpression := ADR(_SqlCommand),			// SQL 命令 ex. SELECT * FROM PlcTest.newtable WHERE ID = {ID}  
				cbExpression := SIZEOF(_SqlCommand),		// SQL 命令字串的長度
				pData:= ADR(Write_Time_para),							// 帶入的參數值
				cbData:= SIZEOF(Write_Time_para),						// 帶入的參數值大小
				pParameter:= ADR(_stPara), 					// 帶入的參數類型設定  ex.上面命令內的 {ID} 類型設定
				cbParameter:= SIZEOF(_stPara[0]) * 2		// 帶入的參數類型設定的大小
			) 
		THEN
			IF MsgMain._fb_PLCDBCmdEvt.bError THEN
				tcMessage := MsgMain._fb_PLCDBCmdEvt.ipTcResult;
				step := step + 10000;
			ELSE
				step := step + 1;
			END_IF
			
		END_IF
	
		
	2012:
		bDone := _sn_cnt1;
		step := 0;

END_CASE
END_ACTION

ACTION Stap_2100_Set_Payload_Finish:
(*	=================================================================
						從資料庫讀取 A頭 雷射檔
	================================================================= *)
CASE step OF
	2100:
		// SQL命令
		_SqlCommand := 
		'SELECT EXISTS(
			SELECT 
				data_uuid
			from 
				public.payloaddata
			where 
				data_uuid = {uuid}::uuid
		);';
				
		
	
		// 設定對應參數
		_stPara[0].sParaName := 'uuid'; 			_stPara[0].eParaType := E_ExpParameterType.STRING_; 		_stPara[0].nParaSize := 37;
		
		step := step + 1;
		
	2101:
		IF 
			MsgMain._fb_PLCDBCmdEvt.ExecuteDataReturn(
				hDBID := database_server_id,
				pExpression := ADR(_SqlCommand),			// SQL 命令 ex. SELECT * FROM PlcTest.newtable WHERE ID = {ID}  
				cbExpression := SIZEOF(_SqlCommand),		// SQL 命令字串的長度
				pData:= ADR(_uuid),							// 帶入的參數值
				cbData:= SIZEOF(_uuid),						// 帶入的參數值大小
				pParameter:= ADR(_stPara), 					// 帶入的參數類型設定  ex.上面命令內的 {ID} 類型設定
				cbParameter:= SIZEOF(_stPara[0]),		// 帶入的參數類型設定的大小
				nStartIndex := 0,
				nRecordCount := 1,
				pReturnData := ADR(_DataExists),
				cbReturnData := SIZEOF(_DataExists),
				pRecords := ADR(read_num)
			) 
		THEN
			IF MsgMain._fb_PLCDBCmdEvt.bError THEN
				tcMessage := MsgMain._fb_PLCDBCmdEvt.ipTcResult;
				step := step + 10000;
			ELSE
				step := step + 1;
			END_IF
			
		END_IF
		
	2102:
		IF _DataExists THEN
			step := step + 1;
		ELSE
			pmsg.Push_Alarm_NoPause(WStrConcat(str0:= "ReadSQLData.Set_Payload_Finish: 讀取的UUID(", str1:= TO_WSTRING(_uuid), str2:= ")不存在。", str3:= TO_WSTRING(step)));
			step := step + 10000;
		END_IF
		
	2103:
			step := 2110;
			
	2110:
		Write_Time_para.Start_TIME := currentTime;
		Write_Time_para.Uid := _uuid;
	
		// SQL命令
		_SqlCommand := 
		'
		UPDATE 
			public.payloaddata 
		SET 
			stage_finish = {timestamp}, is_stage_finish = true
		WHERE
			data_uuid = {id}::UUID
		';
		
	
		// 設定對應參數
		_stPara[0].sParaName := 'timestamp'; 			_stPara[0].eParaType := E_ExpParameterType.DateTime; 		_stPara[0].nParaSize := SIZEOF(Write_Time_para.Start_TIME);
		_stPara[1].sParaName := 'id'; 					_stPara[1].eParaType := E_ExpParameterType.STRING_; 		_stPara[1].nParaSize := 37;
		
		step := step + 1;
		
	2111:
		IF 
			MsgMain._fb_PLCDBCmdEvt.Execute(
				hDBID := database_server_id,
				pExpression := ADR(_SqlCommand),			// SQL 命令 ex. SELECT * FROM PlcTest.newtable WHERE ID = {ID}  
				cbExpression := SIZEOF(_SqlCommand),		// SQL 命令字串的長度
				pData:= ADR(Write_Time_para),							// 帶入的參數值
				cbData:= SIZEOF(Write_Time_para),						// 帶入的參數值大小
				pParameter:= ADR(_stPara), 					// 帶入的參數類型設定  ex.上面命令內的 {ID} 類型設定
				cbParameter:= SIZEOF(_stPara[0]) * 2		// 帶入的參數類型設定的大小
			) 
		THEN
			IF MsgMain._fb_PLCDBCmdEvt.bError THEN
				tcMessage := MsgMain._fb_PLCDBCmdEvt.ipTcResult;
				step := step + 10000;
			ELSE
				step := step + 1;
			END_IF
			
		END_IF
	
		
	2112:
		bDone := _sn_cnt1;
		step := 0;

END_CASE
END_ACTION

ACTION Stap_3000_Set_Steel_Start:
(*	=================================================================
						寫入 steel 加工開始時間
	================================================================= *)
CASE step OF
	3000:
		// SQL命令
		_SqlCommand := 
		'SELECT EXISTS(
			SELECT 
				part_nest_id
			from 
				public.work_order_data
			where 
				part_nest_id = {uuid}
		);';
				
		
	
		// 設定對應參數
		_stPara[0].sParaName := 'uuid'; 			_stPara[0].eParaType := E_ExpParameterType.STRING_; 		_stPara[0].nParaSize := 37;
		
		step := step + 1;
		
	3001:
		IF 
			MsgMain._fb_PLCDBCmdEvt.ExecuteDataReturn(
				hDBID := database_server_id,
				pExpression := ADR(_SqlCommand),			// SQL 命令 ex. SELECT * FROM PlcTest.newtable WHERE ID = {ID}  
				cbExpression := SIZEOF(_SqlCommand),		// SQL 命令字串的長度
				pData:= ADR(_uuid),							// 帶入的參數值
				cbData:= SIZEOF(_uuid),						// 帶入的參數值大小
				pParameter:= ADR(_stPara), 					// 帶入的參數類型設定  ex.上面命令內的 {ID} 類型設定
				cbParameter:= SIZEOF(_stPara[0]),		// 帶入的參數類型設定的大小
				nStartIndex := 0,
				nRecordCount := 1,
				pReturnData := ADR(_DataExists),
				cbReturnData := SIZEOF(_DataExists),
				pRecords := ADR(read_num)
			) 
		THEN
			IF MsgMain._fb_PLCDBCmdEvt.bError THEN
				tcMessage := MsgMain._fb_PLCDBCmdEvt.ipTcResult;
				step := step + 10000;
			ELSE
				step := step + 1;
			END_IF
			
		END_IF
		
	3002:
		IF _DataExists THEN
			step := step + 1;
		ELSE
			pmsg.Push_Alarm(WStrConcat(str0:= "ReadSQLData.Set_Steel_Start: 讀取的UUID(", str1:= TO_WSTRING(_uuid), str2:= ")不存在。", str3:= TO_WSTRING(step)));
		END_IF
		
	3003:
			step := 3010;
			
	3010:
		Write_Time_para.Start_TIME := currentTime;
		Write_Time_para.Uid := _uuid;
	
		// SQL命令
		_SqlCommand := 
		'
		UPDATE 
			public.work_order_data 
		SET 
			steel_status = $'machining$', steel_location = $'machine$'
		WHERE
			part_nest_id = {id}
		';
		
	
		// 設定對應參數
		_stPara[0].sParaName := 'id'; 			_stPara[0].eParaType := E_ExpParameterType.STRING_; 		_stPara[0].nParaSize := 37;
		
		step := step + 1;
		
	3011:
		IF 
			MsgMain._fb_PLCDBCmdEvt.Execute(
				hDBID := database_server_id,
				pExpression := ADR(_SqlCommand),			// SQL 命令 ex. SELECT * FROM PlcTest.newtable WHERE ID = {ID}  
				cbExpression := SIZEOF(_SqlCommand),		// SQL 命令字串的長度
				pData:= ADR(_uuid),							// 帶入的參數值
				cbData:= SIZEOF(_uuid),						// 帶入的參數值大小
				pParameter:= ADR(_stPara), 					// 帶入的參數類型設定  ex.上面命令內的 {ID} 類型設定
				cbParameter:= SIZEOF(_stPara[0])		// 帶入的參數類型設定的大小
			) 
		THEN
			IF MsgMain._fb_PLCDBCmdEvt.bError THEN
				tcMessage := MsgMain._fb_PLCDBCmdEvt.ipTcResult;
				step := step + 10000;
			ELSE
				step := step + 1;
			END_IF
			
		END_IF
	
		
	3012:
		pMsg.Push_Info(WStrConcat(
				"Set_Steel_Start: ",
				WLEFT(STR:= TO_WSTRING(_uuid), SIZE:= 8),
				" :狀態設定為:加工中(machining), "
				));
		step := 3020;	


	3020:
		// SQL命令
		_SqlCommand := 
		'SELECT EXISTS(
			SELECT 
				id
			from 
				public.steeldata
			where 
				id = {uuid}::uuid
		);';
				
		
	
		// 設定對應參數
		_stPara[0].sParaName := 'uuid'; 			_stPara[0].eParaType := E_ExpParameterType.STRING_; 		_stPara[0].nParaSize := 37;
		
		step := step + 1;
		
	3021:
		IF 
			MsgMain._fb_PLCDBCmdEvt.ExecuteDataReturn(
				hDBID := database_server_id,
				pExpression := ADR(_SqlCommand),			// SQL 命令 ex. SELECT * FROM PlcTest.newtable WHERE ID = {ID}  
				cbExpression := SIZEOF(_SqlCommand),		// SQL 命令字串的長度
				pData:= ADR(_uuid),							// 帶入的參數值
				cbData:= SIZEOF(_uuid),						// 帶入的參數值大小
				pParameter:= ADR(_stPara), 					// 帶入的參數類型設定  ex.上面命令內的 {ID} 類型設定
				cbParameter:= SIZEOF(_stPara[0]),		// 帶入的參數類型設定的大小
				nStartIndex := 0,
				nRecordCount := 1,
				pReturnData := ADR(_DataExists),
				cbReturnData := SIZEOF(_DataExists),
				pRecords := ADR(read_num)
			) 
		THEN
			IF MsgMain._fb_PLCDBCmdEvt.bError THEN
				tcMessage := MsgMain._fb_PLCDBCmdEvt.ipTcResult;
				step := step + 10000;
			ELSE
				step := step + 1;
			END_IF
			
		END_IF
		
	3022:
		IF _DataExists THEN
			step := step + 1;
		ELSE
			pmsg.Push_Alarm(WStrConcat(str0:= "ReadSQLData.Get_DxfData: 讀取的UUID(", str1:= TO_WSTRING(_uuid), str2:= ")不存在。", str3:= TO_WSTRING(step)));
		END_IF
		
	3023:
			step := 3030;
			
	3030:
		Write_Time_para.Start_TIME := currentTime;
		Write_Time_para.Uid := _uuid;
	
		// SQL命令
		_SqlCommand := 
		'
		UPDATE 
			public.steeldata 
		SET 
			job_start_time = {timestamp}
		WHERE
			id = {id}::UUID
		';
		
	
		// 設定對應參數
		_stPara[0].sParaName := 'timestamp'; 			_stPara[0].eParaType := E_ExpParameterType.DateTime; 		_stPara[0].nParaSize := SIZEOF(Write_Time_para.Start_TIME);
		_stPara[1].sParaName := 'id'; 					_stPara[1].eParaType := E_ExpParameterType.STRING_; 		_stPara[1].nParaSize := 37;
		
		step := step + 1;
		
	3031:
		IF 
			MsgMain._fb_PLCDBCmdEvt.Execute(
				hDBID := database_server_id,
				pExpression := ADR(_SqlCommand),			// SQL 命令 ex. SELECT * FROM PlcTest.newtable WHERE ID = {ID}  
				cbExpression := SIZEOF(_SqlCommand),		// SQL 命令字串的長度
				pData:= ADR(Write_Time_para),							// 帶入的參數值
				cbData:= SIZEOF(Write_Time_para),						// 帶入的參數值大小
				pParameter:= ADR(_stPara), 					// 帶入的參數類型設定  ex.上面命令內的 {ID} 類型設定
				cbParameter:= SIZEOF(_stPara[0]) * 2		// 帶入的參數類型設定的大小
			) 
		THEN
			IF MsgMain._fb_PLCDBCmdEvt.bError THEN
				tcMessage := MsgMain._fb_PLCDBCmdEvt.ipTcResult;
				step := step + 10000;
			ELSE
				step := step + 1;
			END_IF
			
		END_IF
	
		
	3032:
		bDone := _sn_cnt1;
		step := 0;

END_CASE
END_ACTION

ACTION Stap_3100_Set_Steel_Finish:
(*	=================================================================
						設定工件完成
	================================================================= *)
CASE step OF
	3100:
		// SQL命令
		_SqlCommand := 
		'SELECT EXISTS(
			SELECT 
				id
			from 
				public.steeldata
			where 
				id = {uuid}::uuid
		);
		';
				
		
	
		// 設定對應參數
		_stPara[0].sParaName := 'uuid'; 			_stPara[0].eParaType := E_ExpParameterType.STRING_; 		_stPara[0].nParaSize := 37;
		
		step := step + 1;
		
	3101:
		IF 
			MsgMain._fb_PLCDBCmdEvt.ExecuteDataReturn(
				hDBID := database_server_id,
				pExpression := ADR(_SqlCommand),			// SQL 命令 ex. SELECT * FROM PlcTest.newtable WHERE ID = {ID}  
				cbExpression := SIZEOF(_SqlCommand),		// SQL 命令字串的長度
				pData:= ADR(_uuid),							// 帶入的參數值
				cbData:= SIZEOF(_uuid),						// 帶入的參數值大小
				pParameter:= ADR(_stPara), 					// 帶入的參數類型設定  ex.上面命令內的 {ID} 類型設定
				cbParameter:= SIZEOF(_stPara[0]),		// 帶入的參數類型設定的大小
				nStartIndex := 0,
				nRecordCount := 1,
				pReturnData := ADR(_DataExists),
				cbReturnData := SIZEOF(_DataExists),
				pRecords := ADR(read_num)
			) 
		THEN
			IF MsgMain._fb_PLCDBCmdEvt.bError THEN
				tcMessage := MsgMain._fb_PLCDBCmdEvt.ipTcResult;
				step := step + 10000;
			ELSE
				step := step + 1;
			END_IF
			
		END_IF
		
	3102:
		IF _DataExists THEN
			step := step + 1;
		ELSE
			pmsg.Push_Alarm(WStrConcat(str0:= "ReadSQLData.Get_DxfData: 讀取的UUID(", str1:= TO_WSTRING(_uuid), str2:= ")不存在。", str3:= TO_WSTRING(step)));
		END_IF
		
	3103:
			step := 3110;
			
	3110:
		Write_Time_para.Start_TIME := currentTime;
		Write_Time_para.Uid := _uuid;
	
		// SQL命令
		_SqlCommand := 
		'
		
		UPDATE 
			public.steeldata 
		SET 
			job_finish_time = {timestamp}, is_job_finish = true
		WHERE
			id = {id}::UUID;
		';
			
		// 設定對應參數
		_stPara[0].sParaName := 'timestamp'; 			_stPara[0].eParaType := E_ExpParameterType.DateTime; 		_stPara[0].nParaSize := SIZEOF(Write_Time_para.Start_TIME);
		_stPara[1].sParaName := 'id'; 					_stPara[1].eParaType := E_ExpParameterType.STRING_; 		_stPara[1].nParaSize := 37;
		
		step := step + 1;
		
	3111:
		IF 
			MsgMain._fb_PLCDBCmdEvt.Execute(
				hDBID := database_server_id,
				pExpression := ADR(_SqlCommand),			// SQL 命令 ex. SELECT * FROM PlcTest.newtable WHERE ID = {ID}  
				cbExpression := SIZEOF(_SqlCommand),		// SQL 命令字串的長度
				pData:= ADR(Write_Time_para),							// 帶入的參數值
				cbData:= SIZEOF(Write_Time_para),						// 帶入的參數值大小
				pParameter:= ADR(_stPara), 					// 帶入的參數類型設定  ex.上面命令內的 {ID} 類型設定
				cbParameter:= SIZEOF(_stPara[0]) * 2		// 帶入的參數類型設定的大小
			) 
		THEN
			IF MsgMain._fb_PLCDBCmdEvt.bError THEN
				tcMessage := MsgMain._fb_PLCDBCmdEvt.ipTcResult;
				step := step + 10000;
			ELSE
				step := step + 1;
			END_IF
			
		END_IF
	
		
	3112:
		step := 3120;
		
	3120:
		// SQL命令
		_SqlCommand := 
		'SELECT EXISTS(
			SELECT 
				part_nest_id
			from 
				public.work_order_data
			where 
				part_nest_id = {uuid}
		);';
				
		
	
		// 設定對應參數
		_stPara[0].sParaName := 'uuid'; 			_stPara[0].eParaType := E_ExpParameterType.STRING_; 		_stPara[0].nParaSize := 37;
		
		step := step + 1;
		
	3121:
		IF 
			MsgMain._fb_PLCDBCmdEvt.ExecuteDataReturn(
				hDBID := database_server_id,
				pExpression := ADR(_SqlCommand),			// SQL 命令 ex. SELECT * FROM PlcTest.newtable WHERE ID = {ID}  
				cbExpression := SIZEOF(_SqlCommand),		// SQL 命令字串的長度
				pData:= ADR(_uuid),							// 帶入的參數值
				cbData:= SIZEOF(_uuid),						// 帶入的參數值大小
				pParameter:= ADR(_stPara), 					// 帶入的參數類型設定  ex.上面命令內的 {ID} 類型設定
				cbParameter:= SIZEOF(_stPara[0]),		// 帶入的參數類型設定的大小
				nStartIndex := 0,
				nRecordCount := 1,
				pReturnData := ADR(_DataExists),
				cbReturnData := SIZEOF(_DataExists),
				pRecords := ADR(read_num)
			) 
		THEN
			IF MsgMain._fb_PLCDBCmdEvt.bError THEN
				tcMessage := MsgMain._fb_PLCDBCmdEvt.ipTcResult;
				step := step + 10000;
			ELSE
				step := step + 1;
			END_IF
			
		END_IF
		
	3122:
		IF _DataExists THEN
			step := step + 1;
		ELSE
			pmsg.Push_Alarm(WStrConcat(str0:= "ReadSQLData.Get_DxfData: 讀取的UUID(", str1:= TO_WSTRING(_uuid), str2:= ")不存在。", str3:= TO_WSTRING(step)));
		END_IF
		
	3123:
			step := 3130;
			
	3130:
		Write_Time_para.Start_TIME := currentTime;
		Write_Time_para.Uid := _uuid;
	
		// SQL命令
		_SqlCommand := 
		'
		UPDATE 
			public.work_order_data 
		SET 
			steel_status = $'finish$', 
			steel_location = $'exitRack$',
			steel_process_is_job_finish = true,
			job_finish_time = {timestamp}
		WHERE
			part_nest_id = {id};
			
		UPDATE 
			public.work_order_data 
		SET 
			sequence_number = sequence_number - 1
		WHERE
			sequence_number > 0;
		';
			
		// 設定對應參數
		_stPara[0].sParaName := 'timestamp'; 			_stPara[0].eParaType := E_ExpParameterType.DateTime; 		_stPara[0].nParaSize := SIZEOF(Write_Time_para.Start_TIME);
		_stPara[1].sParaName := 'id'; 					_stPara[1].eParaType := E_ExpParameterType.STRING_; 		_stPara[1].nParaSize := 37;
		step := step + 1;
		
	3131:
		IF 
			MsgMain._fb_PLCDBCmdEvt.Execute(
				hDBID := database_server_id,
				pExpression := ADR(_SqlCommand),			// SQL 命令 ex. SELECT * FROM PlcTest.newtable WHERE ID = {ID}  
				cbExpression := SIZEOF(_SqlCommand),		// SQL 命令字串的長度
				pData:= ADR(Write_Time_para),							// 帶入的參數值
				cbData:= SIZEOF(Write_Time_para),						// 帶入的參數值大小
				pParameter:= ADR(_stPara), 					// 帶入的參數類型設定  ex.上面命令內的 {ID} 類型設定
				cbParameter:= SIZEOF(_stPara[0])*2			// 帶入的參數類型設定的大小
			) 
		THEN
			IF MsgMain._fb_PLCDBCmdEvt.bError THEN
				tcMessage := MsgMain._fb_PLCDBCmdEvt.ipTcResult;
				step := step + 10000;
			ELSE
				step := step + 1;
			END_IF
			
		END_IF
	
		
	3132:
		pMsg.Push_Info(WStrConcat(
				"Set_Steel_Start: ",
				WLEFT(STR:= TO_WSTRING(_uuid), SIZE:= 8),
				" :狀態設定為:完成(finish), "
				));
		step := 3200;

END_CASE
END_ACTION

ACTION Stap_3200_Set_Steel_SN:
(*	=================================================================
						從資料庫讀取 A頭 雷射檔
	================================================================= *)
CASE step OF
	3200: 
		step := 3220;


	3220:
		// SQL命令
		_SqlCommand := 
		'
		UPDATE
			public.work_order_data
		SET 
			sequence_number = sequence_number - 1
		WHERE
			sequence_number > 1
		
		';

		step := step + 1;
		
	3221:
		IF 
			MsgMain._fb_PLCDBCmdEvt.Execute(
				hDBID := database_server_id,
				pExpression := ADR(_SqlCommand),			// SQL 命令 ex. SELECT * FROM PlcTest.newtable WHERE ID = {ID}  
				cbExpression := SIZEOF(_SqlCommand),		// SQL 命令字串的長度
				pData:= 0,							// 帶入的參數值
				cbData:= 0,						// 帶入的參數值大小
				pParameter:= 0, 					// 帶入的參數類型設定  ex.上面命令內的 {ID} 類型設定
				cbParameter:= 0			// 帶入的參數類型設定的大小
			) 
		THEN
			IF MsgMain._fb_PLCDBCmdEvt.bError THEN
				tcMessage := MsgMain._fb_PLCDBCmdEvt.ipTcResult;
				step := step + 10000;
			ELSE
				step := step + 1;
			END_IF
			
		END_IF
	
		
	3222:
		step := 3230;
		
	3230:
		bDone := _sn_cnt1;
		step := 0;

END_CASE
END_ACTION

END_PROGRAM

// ---- MSG/通知訊息/MsgMain.TcPOU
PROGRAM MsgMain
VAR
	
	
	MsgNum			: USINT;
	
	_fb_PLCDBCmdEvt : FB_PLCDBCmdEvt(sNetID:= '', tTimeout:= T#5S );
	
	msg		: MsgStruct;
	
	_SqlCommand : STRING(255);
	
	_stPara		: ARRAY [0..5] OF ST_ExpParameter;
	
	tcMessage     : I_TcMessage;
	
	itmp: UINT;
	
	msgtmp		: MsgStruct_RAW;
	
	str : POINTER TO ARRAY[0..159] OF BYTE;
	
	str2 : POINTER TO ARRAY[0..159] OF BYTE;
	
	str3 : POINTER TO ARRAY[0..499] OF BYTE;
END_VAR

IF msgbuff.DoneNumber < msgbuff.evenNumber THEN
	MsgNum := ULINT_TO_USINT(msgbuff.DoneNumber MOD 16);

	msg := msgbuff.messageList[MsgNum];

	// SQL命令
	_SqlCommand := 
//	'INSERT INTO msg (su, msgtime, msg_level, msgnum, str1, str2) VALUES (uuidv7(), {msgtime}, {msg_level}, {msgnum}, {str1})';

	'INSERT INTO msg (su, msgtime, msg_level, msgnum, str1, str2, raw_msg_str) VALUES (uuidv7(), {msgtime}::timestamptz, {msg_level}, {msgnum}, {str1}, {str2}, {raw_msg_str})';

	msgtmp.msgTIME := msg.msgTIME;
	msgtmp.Level := msg.Level;
	msgtmp.Number := msg.Number;

	str := ADR(msg.MsgStr1);
	msgtmp.MsgStr1 := str^;

	str2 := ADR(msg.MsgStr2);
	msgtmp.MsgStr2 := str2^;

	str3 := ADR(msg.raw_msg_str);
	msgtmp.raw_msg_str := str3^;


// 設定對應參數
	_stPara[0].sParaName := 'msgtime'; 		_stPara[0].eParaType := E_ExpParameterType.DateTime; 	_stPara[0].nParaSize := SIZEOF(msgtmp.msgTIME);
	_stPara[1].sParaName := 'msg_level'; 	_stPara[1].eParaType := E_ExpParameterType.Int16; 		_stPara[1].nParaSize := SIZEOF(msgtmp.Level);
	_stPara[2].sParaName := 'msgnum';		_stPara[2].eParaType := E_ExpParameterType.Int16;		_stPara[2].nParaSize := SIZEOF(msgtmp.Number);
	_stPara[3].sParaName := 'str1';			_stPara[3].eParaType := E_ExpParameterType.WSTRING_;	_stPara[3].nParaSize := 160;
	_stPara[4].sParaName := 'str2';			_stPara[4].eParaType := E_ExpParameterType.WSTRING_;	_stPara[4].nParaSize := 160;
	_stPara[5].sParaName := 'raw_msg_str';	_stPara[5].eParaType := E_ExpParameterType.WSTRING_;	_stPara[5].nParaSize := 500;


	IF 
		MsgMain._fb_PLCDBCmdEvt.Execute(
			hDBID := 1,
			pExpression := ADR(_SqlCommand),			// SQL 命令 ex. SELECT * FROM PlcTest.newtable WHERE ID = {ID}  
			cbExpression := SIZEOF(_SqlCommand),		// SQL 命令字串的長度
			pData:= ADR(msgtmp),		// 帶入的參數值
			cbData:= SIZEOF(msgtmp),//itmp, 	// 帶入的參數值大小
			pParameter:= ADR(_stPara), 				// 帶入的參數類型設定  ex.上面命令內的 {ID} 類型設定
			cbParameter:= SIZEOF(_stPara),			// 帶入的參數類型設定的大小
		) 
	THEN
		IF MsgMain._fb_PLCDBCmdEvt.bError THEN
			tcMessage := MsgMain._fb_PLCDBCmdEvt.ipTcResult;
		END_IF
		msgbuff.DoneNumber := msgbuff.DoneNumber + 1;
	END_IF
ELSIF msgbuff.DoneNumber > msgbuff.evenNumber THEN
	msgbuff.DoneNumber := msgbuff.evenNumber;
END_IF

msgbuff.systime(
	bEnable:= TRUE, 
	dwCycle:= 1,
	systemTime=> );
msgbuff.currentTime := SYSTEMTIME_TO_DT(msgbuff.systime.systemTime);

END_PROGRAM

// ---- POUs/動作流程控制/AxisGroup功能塊/GroupB.TcPOU
PROGRAM GroupB
VAR
	step		: INT;
	
	StepA		: Sub_Step;
	
	// X軸映射
	Ax : I_Axis;
	Axs: Sub_Step;
	// Y軸映射
	Ay : I_Axis;
	Ays: Sub_Step;
	// X軸映射
	Az : I_Axis;
	Azs: Sub_Step;
	
	Ax_P_Limite : LREAL;
	Ax_N_Limite : LREAL;
	Ay_P_Limite : LREAL;
	Ay_N_Limite : LREAL;
	Az_P_Limite : LREAL;
	Az_N_Limite : LREAL;
	
	
	// 移動命令的 X位置
	moveCmd_X: LREAL;
	// 移動命令的 Y位置
	moveCmd_Y: LREAL;
	// 移動命令 速度
	moveCmd_Spd: LREAL;
	
	moveZdis	: REAL;
	tmr01A		: TON;
	tmr01		: TON;
	tmr02		: TON;
	
	// 坐標系的參考原點
	pointRef : XYZ_Point;
	
	// 移動位置X 計算結果
	tmpPos_X: LREAL;
	// 移動位置Y 計算結果
	tmpPos_Y: LREAL;
	
	// 雷射圖形移動距離 Y
	Dxf_Y_Move : LREAL;
	

	// 測量到的Z位置
	z_PosMeasure: REAL;
	
	// 距離感應器IO
	DisSensor_SSC1: BOOL;
	// 距離感應器距離
	DisSensor_Dis: LREAL;
	
	Boot : BOOL := TRUE;
	
	
	
	// 執行中的清單號
	WorkNum: INT;
	
	// 鏡頭 吹氣
	q_Lens_Blow :BOOL;
	
	// 重試計數器
	_retryCnt: INT;
	tmpPos_Z: LREAL;
	
	// 可以開始雕刻 (Fx就緒)
	_ReadyToPrint :BOOL;
	// 可以開始移動 (Fx就緒)
	_ReadyToMove :BOOL;
	
	
	// 計算上次打油後的一棟距離
	X_Move: LREAL;
	Y_Move: LREAL;
	Z_Move: LREAL;
	tmr_oil: TON;
	
	_log : Step_Log; 
	_logA : Step_Log; 
	sql_hand: UDINT;
	tmpPos_Y1: LREAL;
END_VAR

VAR_OUTPUT
	// 工件高度
	Size_H : REAL;
	// 工件座標
	RefPos : XYZ_Point;
	
	// 功能執行中
	bBuzy 	: BOOL;
	// 功能結束
	bDone	: BOOL;
	// 發生錯誤
	bError	: BOOL;
END_VAR

IF Boot THEN
	Ax := axis.GbX;
	Ay := axis.GbY;
	Az := axis.GbZ;
	boot := FALSE;
END_IF

Axs := Ax.State;
Ays := Ay.State;
Azs := Az.State;

Ax_P_Limite := posc.GbX_P_Limite;
Ax_N_Limite := posc.GbX_N_Limite;
Ay_P_Limite := posc.GbY_P_Limite;
Ay_N_Limite := posc.GbY_N_Limite;
Az_P_Limite := posc.GbZ_P_Limite;
Az_N_Limite := posc.GbZ_N_Limite;


DisSensor_SSC1	:= Sensor.sensorB.SSC1_1;
DisSensor_Dis	:= Sensor.sensorB.Distance;

IF (EStop OR SystemError) THEN
	IF bBuzy THEN
		step := step  + 10000;
	END_IF
	IF StepA.bBuzy THEN
		StepA.step := StepA.step  + 10000;
	END_IF
	Hmi_Web.Process_Data_UUID_B_Start := FALSE;
	q_Lens_Blow := FALSE;
END_IF

bBuzy := step > 0 AND step < 10000;
bError := step >= 10000;
IF bBuzy OR bError THEN
	bDone := FALSE;
END_IF

Step_01_DoPayloadList();
Step_02_Do_2nd_in_list();
Step_03_DoLaserAction();



StepA.bBuzy := StepA.step > 0 AND StepA.step < 10000;
StepA.bError := StepA.step >= 10000;
IF StepA.bBuzy OR StepA.bError THEN
	StepA.bDone := FALSE;
END_IF

Step_A_01_MoveToXY();
Step_A_02_FindZ();
Step_A_03_FindY();
Step_A_10_MoveToXY_REF();
Step_A_20_ToStanbyPos();

Timer();

RefPos.X := Ax.Pos + pointRef.X;
RefPos.Y := Ay.Pos - pointRef.Y;
RefPos.Z := Az.Pos - pointRef.Z;

ProjectData.Now_Steel_Payload_B_DataNumberDone := WorkNum;

io.q306 := q_Lens_Blow;

_log(name:= 'GroupB', step:= step);
_logA(name:= 'GroupB_Mov', step:= StepA.Step);

METHOD Do_WorkList : BOOL
VAR_INPUT
END_VAR
bDone := FALSE;

// ============ 紀錄啟動條件 ============
_log.fbJson.StartObject();
_log.fbJson.AddKeyString('MethodName','Do_WorkList');
_log.JsonOutput();
// ======================================



Step := 100;
END_METHOD

METHOD FindZ : BOOL
VAR_INPUT
END_VAR
StepA.bDone := FALSE;

// ============ 紀錄啟動條件 ============
_logA.fbJson.StartObject();
_logA.fbJson.AddKeyString('MethodName','FindZ');
_logA.JsonOutput();
// ======================================






StepA.step := 200;
END_METHOD

METHOD FindZ_Fast : BOOL
VAR_INPUT
END_VAR
StepA.bDone := FALSE;

// ============ 紀錄啟動條件 ============
_logA.fbJson.StartObject();
_logA.fbJson.AddKeyString('MethodName','FindZ_Fast');
_logA.JsonOutput();
// ======================================





StepA.step := 220;
END_METHOD

ACTION Oil:
X_Move := Axis.GbX_total_Move - Axis.GbX_Last_Oil;
Y_Move := Axis.GbY_total_Move - Axis.GbY_Last_Oil;
Z_Move := Axis.GbZ_total_Move - Axis.GbZ_Last_Oil;

IF X_Move > 1000000 OR Y_Move > 1000000 OR Z_Move > 1000000 THEN
	IO.q205 := TRUE;
END_IF
END_ACTION

PROPERTY ReadyToMove : BOOL
GET
ReadyToMove := _ReadyToMove;
END_GET
SET
_ReadyToMove := ReadyToMove;
END_SET
END_PROPERTY

PROPERTY ReadyToPrint : BOOL
GET
ReadyToPrint := _ReadyToPrint;
END_GET
SET
_ReadyToPrint := ReadyToPrint;
END_SET
END_PROPERTY

METHOD Set_X_Ref
VAR_INPUT
	Value : LREAL;
END_VAR
pointRef.X := Value;
END_METHOD

METHOD Set_Y_Ref
VAR_INPUT
	Value : LREAL;
END_VAR
pointRef.Y := Value;
END_METHOD

ACTION Step_01_DoPayloadList:
CASE step OF
(*	===============================================
		開始做 Payload_B_Data_buff 清單內的工作
	===============================================*)
	100: // 以數量判斷是否有工作
		WorkNum := 0;		// 初始化工作暫存器
		IF ProjectData.Now_Steel_Payload_B_DataNumber > 0 THEN
			step := step + 1;
		ELSE
		// 沒有這個軸向的工作，直接送出完成
			bDone := TRUE;
			Step := 0;
		END_IF
 
			
	101:
		Hmi_Web.Process_Data_UUID_B_Start := FALSE;
		step := 110;
		
(*	===============================================
					設定工作中的專案
	===============================================*)
	110:
		ProjectData.Payload_B_Data_Now := ProjectData.Payload_B_Data_buff[WorkNum];
		Hmi_Web.Process_Data_UUID_B := ProjectData.Payload_B_Data_buff[WorkNum].data_uid;
		step := step + 1;
	
	111:
		step := 120;
		
(*	===============================================
					移動到位置
	===============================================*)
	120:
		IF _ReadyToMove THEN
			step := step + 1;
		END_IF
		
	121:
		tmpPos_Y1 := ProjectData.Payload_B_Data_Now.Point_Y;
		
// 		IF tmpPos_Y1 > 80 AND tmpPos_Y1 < (ProjectData.Now_Steel.Height -80) THEN
// 			tmpPos_Y1 := tmpPos_Y1 - 2;
// 		END_IF
		
		XY_Move_Ref(
			ProjectData.Payload_B_Data_Now.Point_X, 
			tmpPos_Y1, 
			SpdC.HighSpeed
		);
		step := step + 1;
		
	122:
		IF stepA.bBuzy OR stepA.bError THEN
			step := step + 1;
		END_IF
		
	123:
		IF stepA.bDone THEN
			step := step + 1;
		ELSIF stepA.bError THEN
			step := step + 10000;
		END_IF
		
	124:
		step := 130;
	

(*	===============================================
				雷射主機 啟動 預覽/雕刻 動作
	===============================================*)	
	130:
		step := 300;
END_CASE
END_ACTION

ACTION Step_02_Do_2nd_in_list:
CASE step OF
	200:
		step := 210;
		
(*	===============================================
					設定工作中的專案
	===============================================*)
	210:
		ProjectData.Payload_B_Data_Now := ProjectData.Payload_B_Data_buff[WorkNum];
		Hmi_Web.Process_Data_UUID_B := ProjectData.Payload_B_Data_buff[WorkNum].data_uid;
		step := step + 1;
	
	211:
		step := 220;
		
(*	===============================================
					移動到位置
	===============================================*)
	220:
		tmpPos_Y1 := ProjectData.Payload_B_Data_Now.Point_Y;
		
// 		IF tmpPos_Y1 > 76 AND tmpPos_Y1 < (ProjectData.Now_Steel.Height - 76) THEN
// 			tmpPos_Y1 := tmpPos_Y1 - 1.5;
// 		END_IF
	
		XY_Move_Ref(
			ProjectData.Payload_B_Data_Now.Point_X, 
			tmpPos_Y1, 
			SpdC.HighSpeed
		);
		step := step + 1;
		
	221:
		IF stepA.bBuzy OR stepA.bError THEN
			step := step + 1;
		END_IF
		
	222:
		IF stepA.bDone THEN
			step := step + 1;
		ELSIF stepA.bError THEN
			step := step + 10000;
		END_IF
		
	223:
		step := 230;

(*	===============================================
				雷射主機 啟動 預覽/雕刻 動作
	===============================================*)	
	230:
		step := 300;
		
END_CASE
END_ACTION

ACTION Step_03_DoLaserAction:
CASE step OF
	300:
		IF ReadyToPrint THEN
			step := step + 1;
		END_IF
		
	301:
		sql_hand := ReadSQLData.Set_Payload_Start(ProjectData.Payload_B_Data_Now.data_uid);
		IF sql_hand <> 0 THEN
			step := step + 1;
		END_IF
		
	302:
		step := 310;

(*	===============================================
				雷射主機 啟動 預覽/雕刻 動作
	===============================================*)	
	310:
		q_Lens_Blow := TRUE;
		IF LEN(Hmi_Web.Process_Data_UUID_B) = 0 THEN
			Hmi_Web.Process_Data_UUID_B := ProjectData.Payload_B_Data_buff[WorkNum].data_uid;
		ELSE
			step := step + 1;
		END_IF
		
	311:
		Hmi_Web.Process_Data_UUID_B_Start := TRUE;
		// ============ 紀錄啟動條件 ============
		_log.fbJson.StartObject();
		_log.fbJson.AddKeyString('StepName','Laser_B_Start');
		_log.fbJson.AddKeyBool('Process_Data_UUID_B_Start:', Hmi_Web.Process_Data_UUID_B_Start);
		_log.fbJson.AddKeyString('Payload_B_Data_Now', ProjectData.Payload_B_Data_Now.data_uid);
		_log.JsonOutput();
		// ======================================
		step := step + 1;
		
	312:	
		tmr01.PT := T#500MS;
		tmr01.IN := TRUE;
		IF tmr01.Q THEN
			tmr01.IN := FALSE;
			tmr02.IN := FALSE;
			step := step + 1;
		END_IF
		
	313:
		tmr01.PT := TO_TIME(MaCfg.LaserPrinter_Timeout);
		tmr01.IN := TRUE;
		tmr02.PT := T#250mS;
		tmr02.IN := NOT Hmi_Web.Process_Data_UUID_B_Start;
		IF tmr02.Q THEN
			Hmi_Web.Process_Data_UUID_B :='';
			tmr01.IN := FALSE;
			tmr02.IN := FALSE;
			// ============ 紀錄啟動條件 ============
			_log.fbJson.StartObject();
			_log.fbJson.AddKeyString('StepName','Laser_B_Done');
			_log.JsonOutput();
			// ======================================
			step := step + 1;
		ELSIF tmr01.Q THEN
			tmr01.IN := FALSE;
			tmr02.IN := FALSE;
			pMsg.Push_Error("GroupB:雷射動作超時");
			step := step + 10000;
		END_IF
	
	314:
		q_Lens_Blow := FALSE;
		WorkNum := WorkNum + 1;
		step := 320;
		
(*	================================================
				開始下個循環或此區域結束
	================================================*)	
	320:
		sql_hand := ReadSQLData.Set_Payload_Finish(ProjectData.Payload_B_Data_Now.data_uid);
		IF sql_hand <> 0 THEN
			step := step + 1;
		END_IF
	
	321:
		IF WorkNum < ProjectData.Now_Steel_Payload_B_DataNumber THEN
		// 這個區域還有工作
			step := step + 1;
		ELSE
		// 這個區域工作結束
			step := 390;
		END_IF
		
	322:
		// 設定工作中的專案
		step := 200;
		
(*	================================================
				此區域結束
	================================================*)		
	390:
		bDone := TRUE;
		step := 0;
END_CASE
END_ACTION

